C07234=1040.428,9.851,-82.657,169.408,37.411,157.036
C07235=1040.433,10.101,-82.672,169.410,37.411,157.036
C07236=1040.440,10.351,-82.687,169.412,37.412,157.036
C07237=1040.446,10.600,-82.703,169.414,37.412,157.036
C07238=1040.453,10.849,-82.718,169.416,37.413,157.036
C07239=1040.460,11.098,-82.734,169.417,37.414,157.036
C07240=1040.466,11.348,-82.749,169.419,37.414,157.037
C07241=1040.472,11.598,-82.764,169.421,37.415,157.037
C07242=1040.479,11.847,-82.779,169.423,37.415,157.037
C07243=1040.485,12.097,-82.795,169.426,37.416,157.037
C07244=1040.492,12.382,-82.812,169.429,37.416,157.037
C07245=1040.500,12.667,-82.830,169.431,37.418,157.037
C07246=1040.507,12.952,-82.848,169.433,37.418,157.037
C07247=1040.514,13.238,-82.865,169.435,37.419,157.038
C07248=1040.521,13.487,-82.880,169.437,37.419,157.038
C07249=1040.528,13.737,-82.895,169.439,37.420,157.038
C07250=1040.534,13.986,-82.911,169.441,37.421,157.038
C07251=1040.540,14.236,-82.927,169.443,37.421,157.038
C07252=1040.547,14.485,-82.942,169.446,37.422,157.038
C07253=1040.553,14.735,-82.957,169.448,37.423,157.039
C07254=1040.559,14.984,-82.973,169.450,37.424,157.039
C07255=1040.566,15.233,-82.989,169.452,37.424,157.039
C07256=1040.574,15.563,-83.009,169.454,37.425,157.039
C07257=1040.582,15.892,-83.031,169.457,37.426,157.039
C07258=1040.590,16.223,-83.051,169.459,37.427,157.039
C07259=1040.599,16.552,-83.071,169.463,37.428,157.040
C07260=1040.605,16.802,-83.087,169.465,37.429,157.040
C07261=1040.611,17.051,-83.103,169.467,37.430,157.040
C07262=1040.618,17.301,-83.118,169.468,37.430,157.040
C07263=1040.624,17.550,-83.134,169.470,37.431,157.040
C07264=1040.630,17.799,-83.150,169.472,37.432,157.040
C07265=1040.637,18.049,-83.165,169.474,37.433,157.041
C07266=1040.643,18.298,-83.181,169.476,37.433,157.041
C07267=1040.649,18.547,-83.197,169.478,37.434,157.041
C07268=1040.656,18.797,-83.212,169.480,37.434,157.041
C07269=1040.662,19.047,-83.228,169.483,37.435,157.041
C07270=1040.669,19.296,-83.244,169.485,37.436,157.041
C07271=1040.675,19.546,-83.260,169.487,37.437,157.041
C07272=1040.681,19.795,-83.275,169.489,37.437,157.042
C07273=1040.688,20.044,-83.291,169.490,37.438,157.042
C07274=1040.694,20.293,-83.307,169.492,37.439,157.042
C07275=1040.700,20.543,-83.323,169.494,37.440,157.042
C07276=1040.706,20.792,-83.338,169.496,37.440,157.042
C07277=1040.712,21.041,-83.355,169.498,37.441,157.042
C07278=1040.720,21.291,-83.371,169.501,37.442,157.042
C07279=1040.725,21.541,-83.386,169.503,37.443,157.043
C07280=1040.732,21.790,-83.402,169.505,37.443,157.043
C07281=1040.738,22.040,-83.418,169.506,37.444,157.043
C07282=1040.745,22.289,-83.434,169.508,37.445,157.043
C07283=1040.750,22.538,-83.450,169.510,37.446,157.043
C07284=1040.757,22.787,-83.466,169.512,37.447,157.043
C07285=1040.763,23.037,-83.481,169.514,37.447,157.044
C07286=1040.770,23.287,-83.497,169.517,37.448,157.044
C07287=1040.776,23.536,-83.514,169.519,37.449,157.044
C07288=1040.782,23.785,-83.530,169.521,37.450,157.044
C07289=1040.789,24.034,-83.545,169.523,37.450,157.044
C07290=1040.795,24.284,-83.562,169.524,37.451,157.044
C07291=1040.801,24.533,-83.577,169.526,37.452,157.045
C07292=1040.808,24.783,-83.593,169.528,37.453,157.045
C07293=1040.814,25.032,-83.609,169.530,37.453,157.045
C07294=1040.820,25.282,-83.625,169.532,37.454,157.045
C07295=1040.827,25.531,-83.641,169.535,37.455,157.045
C07296=1040.833,25.780,-83.657,169.537,37.456,157.045
C07297=1040.839,26.030,-83.674,169.539,37.456,157.046
C07298=1040.846,26.279,-83.689,169.540,37.457,157.046
C07299=1040.852,26.529,-83.706,169.542,37.458,157.046
C07300=1040.859,26.778,-83.721,169.544,37.459,157.046
C07301=1040.865,27.027,-83.738,169.546,37.459,157.046
C07302=1040.871,27.277,-83.754,169.548,37.460,157.046
C07303=1040.878,27.526,-83.770,169.551,37.461,157.047
C07304=1040.883,27.754,-83.785,169.552,37.462,157.047
C07305=1040.889,27.982,-83.799,169.554,37.462,157.047
C07306=1040.895,28.210,-83.814,169.556,37.463,157.047
C07307=1040.901,28.438,-83.829,169.558,37.463,157.047
C07308=1040.906,28.666,-83.843,169.559,37.464,157.047
C07309=1040.912,28.893,-83.858,169.561,37.465,157.047
C07310=1040.918,29.122,-83.873,169.563,37.466,157.048
C07311=1040.924,29.350,-83.888,169.564,37.466,157.048
C07312=1040.930,29.599,-83.905,169.566,37.467,157.048
C07313=1040.936,29.848,-83.921,169.569,37.468,157.048
C07314=1040.942,30.097,-83.937,169.571,37.469,157.048
C07315=1040.949,30.347,-83.953,169.573,37.469,157.048
C07316=1040.955,30.597,-83.969,169.575,37.471,157.049
C07317=1040.961,30.846,-83.986,169.576,37.471,157.049
C07318=1040.967,31.095,-84.002,169.578,37.472,157.049
C07319=1040.974,31.345,-84.019,169.580,37.473,157.049
C07320=1040.980,31.594,-84.034,169.583,37.474,157.049
C07321=1040.987,31.843,-84.051,169.585,37.474,157.049
C07322=1040.993,32.092,-84.068,169.587,37.475,157.050
C07323=1040.999,32.342,-84.084,169.588,37.476,157.050
C07324=1041.006,32.592,-84.100,169.590,37.477,157.050
C07325=1041.012,32.841,-84.116,169.592,37.478,157.050
C07326=1041.018,33.091,-84.133,169.594,37.478,157.050
C07327=1041.025,33.340,-84.150,169.596,37.479,157.050
C07328=1041.031,33.589,-84.166,169.599,37.480,157.051
C07329=1041.037,33.838,-84.182,169.600,37.481,157.051
C07330=1041.044,34.088,-84.198,169.602,37.481,157.051
C07331=1041.050,34.337,-84.214,169.604,37.483,157.051
C07332=1041.056,34.586,-84.231,169.606,37.483,157.051
C07333=1041.063,34.836,-84.248,169.608,37.484,157.051
C07334=1041.069,35.086,-84.264,169.610,37.485,157.052
C07335=1041.075,35.335,-84.280,169.612,37.486,157.052
C07336=1041.082,35.584,-84.297,169.613,37.486,157.052
C07337=1041.088,35.833,-84.314,169.616,37.487,157.052
C07338=1041.094,36.083,-84.330,169.618,37.488,157.052
C07339=1041.101,36.333,-84.346,169.620,37.489,157.052
C07340=1041.107,36.582,-84.363,169.622,37.489,157.053
C07341=1041.114,36.831,-84.379,169.624,37.490,157.053
C07342=1041.120,37.081,-84.396,169.625,37.491,157.053
C07343=1041.126,37.330,-84.412,169.627,37.492,157.053
C07344=1041.133,37.579,-84.429,169.630,37.493,157.053
C07345=1041.139,37.829,-84.446,169.632,37.493,157.053
C07346=1041.145,38.077,-84.463,169.634,37.494,157.054
C07347=1041.152,38.328,-84.479,169.635,37.495,157.054
C07348=1041.158,38.577,-84.495,169.637,37.496,157.054
C07349=1041.164,38.826,-84.512,169.639,37.497,157.054
C07350=1041.170,39.076,-84.529,169.641,37.498,157.054
C07351=1041.176,39.325,-84.545,169.643,37.499,157.055
C07352=1041.183,39.574,-84.562,169.645,37.499,157.055
C07353=1041.189,39.824,-84.579,169.647,37.500,157.055
C07354=1041.195,40.072,-84.596,169.649,37.501,157.055
C07355=1041.202,40.323,-84.612,169.651,37.502,157.055
C07356=1041.208,40.571,-84.629,169.653,37.503,157.056
C07357=1041.214,40.821,-84.646,169.655,37.504,157.056
C07358=1041.220,41.071,-84.663,169.656,37.504,157.056
C07359=1041.226,41.320,-84.680,169.658,37.506,157.056
C07360=1041.233,41.570,-84.696,169.661,37.506,157.056
C07361=1041.239,41.818,-84.713,169.663,37.507,157.056
C07362=1041.245,42.068,-84.730,169.665,37.508,157.057
C07363=1041.252,42.317,-84.747,169.666,37.509,157.057
C07364=1041.258,42.567,-84.763,169.668,37.510,157.057
C07365=1041.265,42.816,-84.781,169.670,37.510,157.057
C07366=1041.271,43.065,-84.797,169.672,37.512,157.057
C07367=1041.277,43.314,-84.814,169.675,37.512,157.057
C07368=1041.284,43.564,-84.831,169.676,37.513,157.058
C07369=1041.289,43.813,-84.848,169.678,37.514,157.058
C07370=1041.296,44.063,-84.865,169.680,37.515,157.058
C07371=1041.302,44.312,-84.882,169.682,37.516,157.058
C07372=1041.309,44.598,-84.902,169.684,37.517,157.058
C07373=1041.316,44.885,-84.921,169.686,37.518,157.059
C07374=1041.323,45.172,-84.940,169.689,37.519,157.059
C07375=1041.330,45.458,-84.961,169.691,37.520,157.059
C07376=1041.336,45.708,-84.977,169.693,37.521,157.059
C07377=1041.342,45.956,-84.994,169.694,37.522,157.059
C07378=1041.349,46.206,-85.012,169.696,37.523,157.060
C07379=1041.355,46.456,-85.028,169.698,37.524,157.060
C07380=1041.361,46.705,-85.046,169.700,37.525,157.060
C07381=1041.367,46.954,-85.063,169.703,37.525,157.060
C07382=1041.373,47.204,-85.080,169.704,37.527,157.060
C07383=1041.380,47.453,-85.097,169.706,37.527,157.061
C07384=1041.386,47.703,-85.115,169.708,37.528,157.061
C07385=1041.392,47.951,-85.132,169.710,37.529,157.061
C07386=1041.399,48.201,-85.148,169.711,37.530,157.061
C07387=1041.404,48.450,-85.166,169.713,37.531,157.061
C07388=1041.410,48.699,-85.183,169.716,37.532,157.062
C07389=1041.417,48.949,-85.199,169.718,37.533,157.062
C07390=1041.422,49.198,-85.217,169.719,37.534,157.062
C07391=1041.429,49.448,-85.234,169.721,37.535,157.062
C07392=1041.436,49.696,-85.251,169.723,37.536,157.062
C07393=1041.441,49.947,-85.268,169.725,37.536,157.063
C07394=1041.448,50.195,-85.285,169.727,37.538,157.063
C07395=1041.455,50.445,-85.303,169.729,37.538,157.063
C07396=1041.460,50.694,-85.320,169.731,37.539,157.063
C07397=1041.467,50.943,-85.338,169.733,37.540,157.063
C07398=1041.473,51.193,-85.354,169.735,37.541,157.064
C07399=1041.479,51.442,-85.372,169.736,37.542,157.064
C07400=1041.486,51.692,-85.389,169.738,37.543,157.064
C07401=1041.492,51.941,-85.406,169.740,37.544,157.064
C07402=1041.498,52.190,-85.424,169.743,37.545,157.064
C07403=1041.504,52.439,-85.441,169.745,37.545,157.064
C07404=1041.510,52.689,-85.458,169.746,37.547,157.065
C07405=1041.517,52.938,-85.475,169.748,37.547,157.065
C07406=1041.523,53.188,-85.493,169.750,37.548,157.065
C07407=1041.529,53.437,-85.510,169.752,37.549,157.065
C07408=1041.536,53.686,-85.528,169.753,37.550,157.065
C07409=1041.543,53.935,-85.545,169.756,37.551,157.066
C07410=1041.548,54.185,-85.562,169.758,37.551,157.066
C07411=1041.555,54.434,-85.580,169.760,37.553,157.066
C07412=1041.561,54.683,-85.597,169.762,37.553,157.066
C07413=1041.567,54.933,-85.614,169.763,37.554,157.066
C07414=1041.574,55.182,-85.631,169.765,37.555,157.066
C07415=1041.579,55.432,-85.649,169.767,37.556,157.067
C07416=1041.586,55.681,-85.666,169.769,37.557,157.067
C07417=1041.593,55.930,-85.683,169.771,37.558,157.067
C07418=1041.599,56.179,-85.701,169.773,37.559,157.067
C07419=1041.606,56.429,-85.718,169.775,37.559,157.067
C07420=1041.612,56.678,-85.735,169.777,37.560,157.068
C07421=1041.618,56.927,-85.753,169.779,37.561,157.068
C07422=1041.625,57.177,-85.771,169.780,37.562,157.068
C07423=1041.630,57.426,-85.788,169.782,37.563,157.068
C07424=1041.637,57.675,-85.806,169.785,37.564,157.068
C07425=1041.643,57.924,-85.823,169.787,37.565,157.069
C07426=1041.650,58.174,-85.840,169.789,37.566,157.069
C07427=1041.656,58.423,-85.858,169.790,37.566,157.069
C07428=1041.662,58.672,-85.875,169.792,37.567,157.069
C07429=1041.669,58.922,-85.893,169.794,37.568,157.069
C07430=1041.676,59.171,-85.910,169.796,37.569,157.069
C07431=1041.682,59.421,-85.928,169.798,37.570,157.070
C07432=1041.688,59.669,-85.945,169.800,37.571,157.070
C07433=1041.694,59.919,-85.963,169.802,37.571,157.070
C07434=1041.701,60.169,-85.980,169.804,37.572,157.070
C07435=1041.707,60.417,-85.997,169.806,37.573,157.070
C07436=1041.715,60.704,-86.018,169.808,37.574,157.071
C07437=1041.722,60.990,-86.037,169.810,37.575,157.071
C07438=1041.730,61.276,-86.059,169.813,37.576,157.071
C07439=1041.737,61.562,-86.078,169.815,37.577,157.071
C07440=1041.743,61.812,-86.096,169.817,37.578,157.071
C07441=1041.750,62.061,-86.114,169.818,37.579,157.072
C07442=1041.756,62.311,-86.131,169.820,37.580,157.072
C07443=1041.762,62.560,-86.149,169.822,37.580,157.072
C07444=1041.769,62.809,-86.166,169.824,37.581,157.072
C07445=1041.775,63.059,-86.184,169.827,37.582,157.072
C07446=1041.782,63.308,-86.202,169.828,37.583,157.073
C07447=1041.788,63.556,-86.219,169.830,37.584,157.073
C07448=1041.794,63.806,-86.237,169.832,37.584,157.073
C07449=1041.801,64.056,-86.255,169.834,37.586,157.073
C07450=1041.807,64.305,-86.272,169.835,37.587,157.073
C07451=1041.813,64.554,-86.290,169.837,37.587,157.073
C07452=1041.819,64.803,-86.308,169.840,37.589,157.074
C07453=1041.826,65.053,-86.326,169.842,37.589,157.074
C07454=1041.832,65.303,-86.344,169.843,37.590,157.074
C07455=1041.838,65.551,-86.362,169.845,37.591,157.074
C07456=1041.845,65.800,-86.379,169.847,37.592,157.074
C07457=1041.851,66.050,-86.397,169.849,37.593,157.075
C07458=1041.858,66.299,-86.416,169.850,37.594,157.075
C07459=1041.864,66.548,-86.433,169.853,37.595,157.075
C07460=1041.870,66.798,-86.451,169.855,37.596,157.075
C07461=1041.876,67.047,-86.469,169.857,37.596,157.075
C07462=1041.883,67.297,-86.487,169.859,37.598,157.076
C07463=1041.889,67.545,-86.504,169.860,37.599,157.076
C07464=1041.895,67.794,-86.523,169.862,37.599,157.076
C07465=1041.901,68.044,-86.541,169.864,37.601,157.076
C07466=1041.907,68.294,-86.559,169.867,37.601,157.076
C07467=1041.914,68.542,-86.576,169.868,37.602,157.077
C07468=1041.920,68.792,-86.594,169.870,37.603,157.077
C07469=1041.926,69.041,-86.612,169.872,37.604,157.077
C07470=1041.933,69.291,-86.631,169.874,37.605,157.077
C07471=1041.940,69.540,-86.648,169.875,37.606,157.077
C07472=1041.945,69.788,-86.667,169.878,37.607,157.078
C07473=1041.951,70.038,-86.685,169.880,37.608,157.078
C07474=1041.958,70.287,-86.703,169.882,37.609,157.078
C07475=1041.964,70.537,-86.721,169.883,37.610,157.078
C07476=1041.970,70.787,-86.739,169.885,37.611,157.078
C07477=1041.976,71.035,-86.757,169.887,37.612,157.079
C07478=1041.983,71.285,-86.775,169.889,37.613,157.079
C07479=1041.989,71.534,-86.793,169.891,37.614,157.079
C07480=1041.995,71.784,-86.811,169.893,37.614,157.079
C07481=1042.002,72.033,-86.830,169.895,37.616,157.079
C07482=1042.007,72.282,-86.847,169.897,37.617,157.080
C07483=1042.014,72.531,-86.866,169.898,37.617,157.080
C07484=1042.020,72.780,-86.885,169.900,37.619,157.080
C07485=1042.026,73.030,-86.903,169.902,37.619,157.080
C07486=1042.033,73.279,-86.921,169.905,37.620,157.080
C07487=1042.038,73.528,-86.939,169.906,37.622,157.081
C07488=1042.045,73.777,-86.958,169.908,37.622,157.081
C07489=1042.052,74.026,-86.975,169.910,37.623,157.081
C07490=1042.058,74.275,-86.994,169.911,37.624,157.081
C07491=1042.064,74.525,-87.012,169.913,37.625,157.081
C07492=1042.070,74.774,-87.030,169.916,37.626,157.082
C07493=1042.077,75.023,-87.049,169.918,37.627,157.082
C07494=1042.082,75.273,-87.066,169.920,37.628,157.082
C07495=1042.089,75.522,-87.085,169.921,37.629,157.082
C07496=1042.095,75.771,-87.104,169.923,37.630,157.083
C07497=1042.101,76.020,-87.122,169.925,37.631,157.083
C07498=1042.108,76.270,-87.140,169.928,37.632,157.083
C07499=1042.114,76.519,-87.158,169.929,37.633,157.083
C07500=1042.122,76.805,-87.179,169.931,37.634,157.083
C07501=1042.128,77.091,-87.200,169.933,37.635,157.084
C07502=1042.136,77.377,-87.222,169.935,37.636,157.084
C07503=1042.143,77.663,-87.243,169.937,37.637,157.084
C07504=1042.149,77.912,-87.261,169.939,37.638,157.084
C07505=1042.155,78.162,-87.279,169.942,37.639,157.084
C07506=1042.162,78.411,-87.298,169.944,37.640,157.085
C07507=1042.168,78.660,-87.316,169.945,37.641,157.085
C07508=1042.174,78.909,-87.335,169.947,37.642,157.085
C07509=1042.180,79.159,-87.354,169.949,37.643,157.085
C07510=1042.186,79.408,-87.372,169.950,37.644,157.085
C07511=1042.193,79.657,-87.391,169.953,37.645,157.086
C07512=1042.199,79.907,-87.409,169.955,37.646,157.086
C07513=1042.205,80.155,-87.427,169.957,37.647,157.086
C07514=1042.210,80.405,-87.447,169.958,37.648,157.086
C07515=1042.217,80.654,-87.465,169.960,37.649,157.087
C07516=1042.223,80.903,-87.484,169.963,37.650,157.087
C07517=1042.229,81.153,-87.502,169.965,37.651,157.087
C07518=1042.236,81.402,-87.520,169.966,37.652,157.087
C07519=1042.242,81.651,-87.540,169.968,37.653,157.088
C07520=1042.248,81.900,-87.558,169.970,37.654,157.088
C07521=1042.254,82.150,-87.577,169.972,37.655,157.088
C07522=1042.261,82.399,-87.596,169.973,37.656,157.088
C07523=1042.267,82.648,-87.614,169.976,37.657,157.088
C07524=1042.273,82.897,-87.634,169.978,37.658,157.089
C07525=1042.279,83.147,-87.651,169.980,37.659,157.089
C07526=1042.285,83.396,-87.670,169.981,37.660,157.089
C07527=1042.291,83.644,-87.688,169.983,37.661,157.089
C07528=1042.298,83.894,-87.707,169.985,37.662,157.089
C07529=1042.303,84.143,-87.726,169.988,37.663,157.090
C07530=1042.310,84.392,-87.745,169.989,37.664,157.090
C07531=1042.316,84.641,-87.764,169.991,37.665,157.090
C07532=1042.323,84.890,-87.782,169.993,37.666,157.090
C07533=1042.329,85.140,-87.801,169.995,37.667,157.091
C07534=1042.335,85.389,-87.820,169.996,37.668,157.091
C07535=1042.341,85.638,-87.839,169.999,37.669,157.091
C07536=1042.348,85.887,-87.857,170.001,37.670,157.091
C07537=1042.354,86.136,-87.876,170.003,37.671,157.091
C07538=1042.360,86.386,-87.895,170.004,37.672,157.092
C07539=1042.366,86.635,-87.914,170.006,37.673,157.092
C07540=1042.373,86.884,-87.933,170.008,37.674,157.092
C07541=1042.380,87.134,-87.952,170.011,37.675,157.092
C07542=1042.386,87.383,-87.970,170.012,37.676,157.092
C07543=1042.392,87.632,-87.990,170.014,37.677,157.093
C07544=1042.398,87.882,-88.008,170.016,37.678,157.093
C07545=1042.405,88.131,-88.027,170.018,37.679,157.093
C07546=1042.411,88.380,-88.045,170.019,37.680,157.093
C07547=1042.417,88.629,-88.065,170.021,37.681,157.093
C07548=1042.423,88.878,-88.083,170.024,37.681,157.094
C07549=1042.430,89.127,-88.102,170.026,37.683,157.094
C07550=1042.436,89.377,-88.121,170.027,37.684,157.094
C07551=1042.442,89.626,-88.140,170.029,37.684,157.094
C07552=1042.448,89.875,-88.159,170.031,37.686,157.095
C07553=1042.455,90.124,-88.177,170.033,37.687,157.095
C07554=1042.460,90.374,-88.196,170.035,37.687,157.095
C07555=1042.467,90.622,-88.216,170.037,37.689,157.095
C07556=1042.473,90.872,-88.235,170.039,37.690,157.095
C07557=1042.480,91.121,-88.254,170.041,37.691,157.096
C07558=1042.485,91.371,-88.273,170.042,37.692,157.096
C07559=1042.492,91.620,-88.292,170.044,37.693,157.096
C07560=1042.498,91.869,-88.312,170.047,37.694,157.096
C07561=1042.504,92.118,-88.331,170.049,37.695,157.097
C07562=1042.510,92.367,-88.350,170.050,37.696,157.097
C07563=1042.516,92.616,-88.368,170.052,37.697,157.097
C07564=1042.524,92.902,-88.391,170.054,37.698,157.097
C07565=1042.531,93.189,-88.412,170.057,37.699,157.097
C07566=1042.537,93.474,-88.435,170.059,37.701,157.098
C07567=1042.544,93.760,-88.457,170.061,37.702,157.098
C07568=1042.551,94.009,-88.475,170.063,37.703,157.098
C07569=1042.557,94.259,-88.496,170.065,37.704,157.099
C07570=1042.564,94.508,-88.514,170.066,37.705,157.099
C07571=1042.569,94.757,-88.534,170.069,37.706,157.099
C07572=1042.576,95.006,-88.552,170.071,37.707,157.099
C07573=1042.582,95.255,-88.572,170.073,37.708,157.099
C07574=1042.588,95.504,-88.591,170.074,37.709,157.100
C07575=1042.594,95.754,-88.610,170.076,37.710,157.100
C07576=1042.600,96.003,-88.630,170.078,37.711,157.100
C07577=1042.607,96.252,-88.649,170.081,37.712,157.100
C07578=1042.613,96.502,-88.668,170.082,37.713,157.100
C07579=1042.619,96.750,-88.688,170.084,37.714,157.101
C07580=1042.625,97.000,-88.707,170.086,37.716,157.101
C07581=1042.631,97.249,-88.725,170.088,37.716,157.101
C07582=1042.637,97.498,-88.745,170.089,37.717,157.101
C07583=1042.644,97.748,-88.764,170.092,37.719,157.102
C07584=1042.650,97.996,-88.784,170.094,37.719,157.102
C07585=1042.657,98.246,-88.803,170.096,37.720,157.102
C07586=1042.662,98.495,-88.822,170.098,37.722,157.102
C07587=1042.668,98.744,-88.842,170.099,37.723,157.103
C07588=1042.675,98.993,-88.861,170.101,37.723,157.103
C07589=1042.682,99.242,-88.881,170.104,37.725,157.103
C07590=1042.688,99.492,-88.900,170.106,37.726,157.103
C07591=1042.694,99.740,-88.920,170.107,37.726,157.103
C07592=1042.700,99.989,-88.938,170.109,37.728,157.104
C07593=1042.706,100.239,-88.958,170.111,37.729,157.104
C07594=1042.713,100.488,-88.978,170.113,37.729,157.104
C07595=1042.719,100.738,-88.997,170.116,37.730,157.104
C07596=1042.725,100.986,-89.017,170.117,37.732,157.104
C07597=1042.731,101.235,-89.037,170.119,37.733,157.105
C07598=1042.737,101.485,-89.056,170.121,37.734,157.105
C07599=1042.743,101.734,-89.076,170.123,37.735,157.105
C07600=1042.750,101.983,-89.095,170.125,37.736,157.105
C07601=1042.756,102.232,-89.115,170.127,37.737,157.106
C07602=1042.761,102.481,-89.134,170.129,37.738,157.106
C07603=1042.767,102.730,-89.154,170.131,37.739,157.106
C07604=1042.774,102.980,-89.174,170.132,37.741,157.106
C07605=1042.780,103.229,-89.193,170.135,37.742,157.107
C07606=1042.786,103.478,-89.213,170.137,37.742,157.107
C07607=1042.792,103.727,-89.232,170.139,37.744,157.107
C07608=1042.798,103.976,-89.252,170.140,37.745,157.107
C07609=1042.805,104.225,-89.272,170.142,37.746,157.108
C07610=1042.811,104.475,-89.291,170.144,37.747,157.108
C07611=1042.817,104.723,-89.311,170.147,37.748,157.108
C07612=1042.823,104.972,-89.331,170.148,37.749,157.108
C07613=1042.829,105.222,-89.351,170.150,37.750,157.108
C07614=1042.835,105.471,-89.371,170.152,37.751,157.109
C07615=1042.841,105.720,-89.391,170.154,37.753,157.109
C07616=1042.848,105.969,-89.409,170.155,37.753,157.109
C07617=1042.854,106.219,-89.430,170.158,37.754,157.109
C07618=1042.860,106.467,-89.449,170.160,37.756,157.110
C07619=1042.866,106.717,-89.469,170.162,37.757,157.110
C07620=1042.873,106.966,-89.489,170.164,37.758,157.110
C07621=1042.879,107.215,-89.509,170.165,37.759,157.110
C07622=1042.885,107.464,-89.528,170.168,37.760,157.111
C07623=1042.891,107.713,-89.548,170.170,37.761,157.111
C07624=1042.898,107.963,-89.568,170.172,37.762,157.111
C07625=1042.904,108.211,-89.588,170.174,37.763,157.111
C07626=1042.909,108.461,-89.607,170.175,37.764,157.111
C07627=1042.916,108.710,-89.627,170.177,37.765,157.112
C07628=1042.923,108.996,-89.650,170.180,37.766,157.112
C07629=1042.930,109.282,-89.673,170.182,37.767,157.112
C07630=1042.938,109.568,-89.695,170.184,37.769,157.113
C07631=1042.944,109.854,-89.718,170.186,37.770,157.113
C07632=1042.951,110.103,-89.738,170.188,37.771,157.113
C07633=1042.957,110.352,-89.758,170.191,37.772,157.113
C07634=1042.963,110.602,-89.779,170.193,37.773,157.114
C07635=1042.970,110.850,-89.798,170.195,37.774,157.114
C07636=1042.975,111.099,-89.819,170.196,37.775,157.114
C07637=1042.982,111.349,-89.838,170.198,37.776,157.114
C07638=1042.988,111.598,-89.858,170.201,37.778,157.114
C07639=1042.994,111.847,-89.878,170.203,37.779,157.115
C07640=1043.000,112.097,-89.898,170.204,37.780,157.115
C07641=1043.006,112.345,-89.918,170.206,37.781,157.115
C07642=1043.012,112.594,-89.938,170.208,37.782,157.115
C07643=1043.019,112.844,-89.959,170.210,37.783,157.116
C07644=1043.025,113.093,-89.979,170.213,37.784,157.116
C07645=1043.031,113.341,-89.999,170.214,37.785,157.116
C07646=1043.037,113.591,-90.019,170.216,37.786,157.116
C07647=1043.043,113.840,-90.039,170.218,37.788,157.117
C07648=1043.049,114.089,-90.059,170.220,37.789,157.117
C07649=1043.056,114.338,-90.079,170.223,37.790,157.117
C07650=1043.061,114.587,-90.100,170.224,37.791,157.117
C07651=1043.067,114.836,-90.120,170.226,37.792,157.118
C07652=1043.074,115.085,-90.140,170.228,37.793,157.118
C07653=1043.079,115.335,-90.161,170.230,37.794,157.118
C07654=1043.085,115.583,-90.181,170.232,37.795,157.118
C07655=1043.092,115.833,-90.201,170.234,37.797,157.119
C07656=1043.098,116.082,-90.221,170.236,37.798,157.119
C07657=1043.104,116.332,-90.242,170.238,37.799,157.119
C07658=1043.110,116.580,-90.262,170.240,37.800,157.119
C07659=1043.116,116.829,-90.282,170.242,37.801,157.120
C07660=1043.122,117.078,-90.303,170.244,37.803,157.120
C07661=1043.128,117.327,-90.323,170.246,37.804,157.120
C07662=1043.134,117.576,-90.343,170.248,37.805,157.120
C07663=1043.140,117.826,-90.364,170.249,37.806,157.121
C07664=1043.146,118.075,-90.384,170.252,37.807,157.121
C07665=1043.152,118.324,-90.404,170.254,37.809,157.121
C07666=1043.158,118.573,-90.424,170.256,37.810,157.121
C07667=1043.164,118.821,-90.445,170.258,37.811,157.122
C07668=1043.170,119.071,-90.466,170.259,37.812,157.122
C07669=1043.176,119.320,-90.486,170.262,37.813,157.122
C07670=1043.183,119.569,-90.506,170.264,37.814,157.123
C07671=1043.188,119.818,-90.527,170.266,37.816,157.123
C07672=1043.195,120.067,-90.548,170.268,37.817,157.123
C07673=1043.201,120.316,-90.568,170.269,37.818,157.123
C07674=1043.206,120.565,-90.588,170.271,37.819,157.123
C07675=1043.213,120.815,-90.609,170.274,37.820,157.124
C07676=1043.219,121.063,-90.629,170.276,37.821,157.124
C07677=1043.225,121.313,-90.650,170.278,37.822,157.124
C07678=1043.231,121.562,-90.670,170.280,37.823,157.124
C07679=1043.238,121.811,-90.691,170.282,37.825,157.125
C07680=1043.244,122.059,-90.711,170.284,37.826,157.125
C07681=1043.250,122.309,-90.732,170.286,37.827,157.125
C07682=1043.256,122.558,-90.752,170.288,37.828,157.126
C07683=1043.262,122.808,-90.772,170.290,37.829,157.126
C07684=1043.268,123.056,-90.794,170.292,37.831,157.126
C07685=1043.275,123.306,-90.814,170.294,37.832,157.126
C07686=1043.281,123.554,-90.834,170.296,37.833,157.127
C07687=1043.287,123.804,-90.856,170.298,37.834,157.127
C07688=1043.293,124.052,-90.876,170.300,37.835,157.127
C07689=1043.299,124.302,-90.896,170.302,37.836,157.127
C07690=1043.305,124.550,-90.917,170.304,37.837,157.127
C07691=1043.311,124.800,-90.937,170.306,37.838,157.128
C07692=1043.318,125.085,-90.961,170.308,37.839,157.128
C07693=1043.326,125.371,-90.985,170.311,37.841,157.128
C07694=1043.333,125.657,-91.008,170.314,37.842,157.129
C07695=1043.340,125.944,-91.032,170.316,37.844,157.129
C07696=1043.346,126.192,-91.053,170.318,37.845,157.129
C07697=1043.353,126.442,-91.074,170.319,37.846,157.129
C07698=1043.359,126.690,-91.094,170.321,37.847,157.130
C07699=1043.365,126.940,-91.115,170.324,37.848,157.130
C07700=1043.371,127.188,-91.135,170.326,37.849,157.130
C07701=1043.378,127.437,-91.156,170.328,37.850,157.130
C07702=1043.383,127.687,-91.177,170.330,37.851,157.131
C07703=1043.390,127.935,-91.198,170.332,37.852,157.131
C07704=1043.396,128.185,-91.219,170.334,37.854,157.131
C07705=1043.402,128.434,-91.239,170.336,37.855,157.131
C07706=1043.409,128.683,-91.260,170.338,37.856,157.132
C07707=1043.414,128.933,-91.281,170.340,37.857,157.132
C07708=1043.421,129.181,-91.301,170.342,37.858,157.132
C07709=1043.427,129.430,-91.322,170.345,37.859,157.132
C07710=1043.433,129.680,-91.343,170.347,37.861,157.133
C07711=1043.439,129.928,-91.363,170.349,37.862,157.133
C07712=1043.446,130.177,-91.384,170.350,37.862,157.133
C07713=1043.452,130.426,-91.406,170.352,37.864,157.133
C07714=1043.458,130.675,-91.426,170.354,37.865,157.134
C07715=1043.465,130.924,-91.448,170.357,37.866,157.134
C07716=1043.471,131.173,-91.468,170.359,37.867,157.134
C07717=1043.477,131.422,-91.489,170.361,37.868,157.134
C07718=1043.483,131.672,-91.510,170.363,37.869,157.135
C07719=1043.489,131.921,-91.531,170.365,37.871,157.135
C07720=1043.495,132.170,-91.552,170.367,37.872,157.135
C07721=1043.502,132.419,-91.573,170.369,37.873,157.135
C07722=1043.507,132.668,-91.594,170.371,37.874,157.136
C07723=1043.513,132.917,-91.616,170.373,37.875,157.136
C07724=1043.519,133.166,-91.636,170.376,37.877,157.136
C07725=1043.526,133.415,-91.657,170.378,37.878,157.137
C07726=1043.532,133.664,-91.679,170.380,37.879,157.137
C07727=1043.538,133.912,-91.700,170.381,37.881,157.137
C07728=1043.544,134.162,-91.720,170.383,37.882,157.137
C07729=1043.550,134.411,-91.742,170.386,37.883,157.138
C07730=1043.556,134.660,-91.763,170.388,37.884,157.138
C07731=1043.563,134.909,-91.784,170.390,37.885,157.138
C07732=1043.568,135.159,-91.805,170.392,37.887,157.138
C07733=1043.575,135.407,-91.826,170.394,37.888,157.139
C07734=1043.581,135.656,-91.848,170.397,37.889,157.139
C07735=1043.587,135.905,-91.869,170.398,37.890,157.139
C07736=1043.593,136.154,-91.889,170.400,37.891,157.140
C07737=1043.599,136.403,-91.911,170.402,37.893,157.140
C07738=1043.605,136.652,-91.933,170.404,37.894,157.140
C07739=1043.612,136.901,-91.954,170.407,37.895,157.140
C07740=1043.618,137.150,-91.975,170.409,37.896,157.141
C07741=1043.624,137.400,-91.996,170.411,37.897,157.141
C07742=1043.630,137.649,-92.017,170.413,37.898,157.141
C07743=1043.636,137.897,-92.038,170.416,37.900,157.141
C07744=1043.642,138.146,-92.060,170.417,37.901,157.142
C07745=1043.648,138.395,-92.081,170.419,37.902,157.142
C07746=1043.655,138.645,-92.103,170.421,37.904,157.142
C07747=1043.660,138.893,-92.124,170.423,37.905,157.143
C07748=1043.667,139.142,-92.145,170.426,37.906,157.143
C07749=1043.673,139.391,-92.167,170.428,37.907,157.143
C07750=1043.679,139.641,-92.188,170.430,37.908,157.143
C07751=1043.685,139.890,-92.209,170.432,37.910,157.144
C07752=1043.691,140.139,-92.231,170.434,37.911,157.144
C07753=1043.697,140.388,-92.252,170.436,37.912,157.144
C07754=1043.703,140.637,-92.274,170.438,37.913,157.144
C07755=1043.709,140.886,-92.295,170.440,37.915,157.145
C07756=1043.717,141.171,-92.320,170.442,37.916,157.145
C07757=1043.723,141.457,-92.344,170.446,37.917,157.145
C07758=1043.730,141.743,-92.370,170.448,37.919,157.146
C07759=1043.737,142.027,-92.394,170.450,37.920,157.146
C07760=1043.744,142.277,-92.416,170.452,37.922,157.146
C07761=1043.750,142.526,-92.437,170.455,37.923,157.147
C07762=1043.756,142.775,-92.459,170.457,37.924,157.147
C07763=1043.761,143.024,-92.480,170.459,37.926,157.147
C07764=1043.768,143.273,-92.502,170.461,37.927,157.147
C07765=1043.774,143.522,-92.523,170.464,37.928,157.148
C07766=1043.780,143.771,-92.545,170.465,37.929,157.148
C07767=1043.786,144.020,-92.567,170.467,37.931,157.148
C07768=1043.792,144.269,-92.588,170.469,37.932,157.149
C07769=1043.798,144.518,-92.610,170.471,37.933,157.149
C07770=1043.804,144.767,-92.632,170.474,37.934,157.149
C07771=1043.810,145.016,-92.654,170.476,37.936,157.149
C07772=1043.817,145.265,-92.675,170.478,37.937,157.150
C07773=1043.823,145.514,-92.697,170.480,37.938,157.150
C07774=1043.828,145.763,-92.718,170.482,37.939,157.150
C07775=1043.835,146.012,-92.740,170.485,37.941,157.151
C07776=1043.841,146.261,-92.761,170.487,37.942,157.151
C07777=1043.847,146.510,-92.784,170.489,37.943,157.151
C07778=1043.854,146.759,-92.805,170.491,37.944,157.151
C07779=1043.860,147.008,-92.826,170.494,37.946,157.152
C07780=1043.865,147.257,-92.848,170.496,37.947,157.152
C07781=1043.871,147.505,-92.871,170.498,37.949,157.152
C07782=1043.878,147.755,-92.892,170.499,37.950,157.153
C07783=1043.884,148.004,-92.914,170.502,37.951,157.153
C07784=1043.890,148.253,-92.936,170.504,37.952,157.153
C07785=1043.896,148.502,-92.958,170.506,37.953,157.153
C07786=1043.903,148.751,-92.980,170.508,37.955,157.154
C07787=1043.909,149.000,-93.001,170.511,37.956,157.154
C07788=1043.914,149.249,-93.023,170.513,37.957,157.154
C07789=1043.920,149.497,-93.045,170.515,37.959,157.155
C07790=1043.926,149.747,-93.067,170.517,37.960,157.155
C07791=1043.933,149.995,-93.089,170.519,37.962,157.155
C07792=1043.939,150.244,-93.111,170.522,37.963,157.155
C07793=1043.945,150.494,-93.133,170.524,37.964,157.156
C07794=1043.951,150.742,-93.156,170.526,37.966,157.156
C07795=1043.957,150.992,-93.177,170.528,37.967,157.156
C07796=1043.963,151.241,-93.199,170.531,37.968,157.157
C07797=1043.969,151.489,-93.221,170.533,37.969,157.157
C07798=1043.975,151.738,-93.242,170.535,37.971,157.157
C07799=1043.981,151.987,-93.265,170.537,37.972,157.158
C07800=1043.987,152.236,-93.287,170.540,37.973,157.158
C07801=1043.993,152.485,-93.309,170.542,37.974,157.158
C07802=1044.000,152.734,-93.331,170.544,37.976,157.158
C07803=1044.005,152.983,-93.353,170.546,37.977,157.159
C07804=1044.012,153.232,-93.376,170.549,37.979,157.159
C07805=1044.018,153.481,-93.397,170.551,37.980,157.159
C07806=1044.024,153.730,-93.420,170.553,37.981,157.160
C07807=1044.030,153.979,-93.441,170.554,37.983,157.160
C07808=1044.036,154.228,-93.464,170.556,37.984,157.160
C07809=1044.042,154.477,-93.486,170.559,37.985,157.160
C07810=1044.049,154.726,-93.508,170.561,37.987,157.161
C07811=1044.054,154.975,-93.530,170.563,37.988,157.161
C07812=1044.061,155.224,-93.553,170.565,37.989,157.161
C07813=1044.067,155.472,-93.575,170.568,37.991,157.162
C07814=1044.072,155.722,-93.597,170.570,37.992,157.162
C07815=1044.079,155.970,-93.620,170.572,37.993,157.162
C07816=1044.085,156.219,-93.641,170.574,37.995,157.163
C07817=1044.090,156.468,-93.664,170.577,37.996,157.163
C07818=1044.097,156.716,-93.686,170.579,37.997,157.163
C07819=1044.102,156.966,-93.708,170.581,37.999,157.164
C07820=1044.110,157.251,-93.735,170.584,38.000,157.164
C07821=1044.117,157.537,-93.760,170.587,38.002,157.164
C07822=1044.124,157.821,-93.786,170.589,38.004,157.165
C07823=1044.131,158.107,-93.811,170.592,38.005,157.165
C07824=1044.137,158.356,-93.834,170.595,38.007,157.165
C07825=1044.143,158.605,-93.855,170.597,38.008,157.166
C07826=1044.149,158.854,-93.878,170.599,38.009,157.166
C07827=1044.155,159.103,-93.901,170.601,38.011,157.166
C07828=1044.161,159.352,-93.922,170.604,38.012,157.167
C07829=1044.168,159.601,-93.945,170.606,38.013,157.167
C07830=1044.173,159.849,-93.968,170.608,38.015,157.167
C07831=1044.180,160.098,-93.990,170.610,38.016,157.167
C07832=1044.185,160.348,-94.012,170.612,38.017,157.168
C07833=1044.192,160.596,-94.035,170.615,38.019,157.168
C07834=1044.198,160.846,-94.058,170.617,38.020,157.168
C07835=1044.204,161.095,-94.081,170.619,38.022,157.169
C07836=1044.209,161.343,-94.104,170.622,38.023,157.169
C07837=1044.215,161.592,-94.127,170.624,38.025,157.169
C07838=1044.222,161.841,-94.149,170.626,38.027,157.170
C07839=1044.227,162.090,-94.171,170.628,38.028,157.170
C07840=1044.233,162.339,-94.194,170.631,38.030,157.171
C07841=1044.239,162.588,-94.217,170.633,38.031,157.171
C07842=1044.245,162.837,-94.240,170.635,38.033,157.171
C07843=1044.251,163.086,-94.263,170.637,38.034,157.171
C07844=1044.256,163.335,-94.285,170.640,38.036,157.172
C07845=1044.262,163.584,-94.308,170.642,38.037,157.172
C07846=1044.268,163.832,-94.331,170.644,38.038,157.173
C07847=1044.274,164.081,-94.354,170.647,38.040,157.173
C07848=1044.280,164.330,-94.377,170.649,38.041,157.173
C07849=1044.286,164.579,-94.400,170.651,38.043,157.174
C07850=1044.292,164.828,-94.423,170.653,38.044,157.174
C07851=1044.297,165.077,-94.446,170.656,38.046,157.174
C07852=1044.304,165.325,-94.468,170.658,38.047,157.175
C07853=1044.310,165.574,-94.491,170.660,38.049,157.175
C07854=1044.315,165.823,-94.514,170.662,38.050,157.175
C07855=1044.321,166.072,-94.537,170.665,38.052,157.176
C07856=1044.327,166.322,-94.560,170.667,38.054,157.176
C07857=1044.334,166.570,-94.582,170.669,38.055,157.176
C07858=1044.340,166.819,-94.605,170.672,38.057,157.177
C07859=1044.345,167.068,-94.628,170.674,38.058,157.177
C07860=1044.351,167.317,-94.651,170.676,38.060,157.177
C07861=1044.357,167.565,-94.675,170.678,38.061,157.178
C07862=1044.363,167.814,-94.698,170.682,38.063,157.178
C07863=1044.369,168.063,-94.720,170.684,38.064,157.178
C07864=1044.376,168.312,-94.743,170.686,38.065,157.179
C07865=1044.381,168.561,-94.766,170.689,38.067,157.179
C07866=1044.387,168.810,-94.789,170.691,38.068,157.179
C07867=1044.393,169.059,-94.812,170.693,38.070,157.180
C07868=1044.400,169.307,-94.835,170.695,38.071,157.180
C07869=1044.405,169.556,-94.858,170.698,38.073,157.180
C07870=1044.412,169.805,-94.882,170.700,38.074,157.181
C07871=1044.417,170.054,-94.905,170.702,38.076,157.181
C07872=1044.423,170.303,-94.928,170.704,38.078,157.181
C07873=1044.429,170.551,-94.951,170.707,38.079,157.182
C07874=1044.435,170.800,-94.974,170.709,38.081,157.182
C07875=1044.442,171.050,-94.997,170.712,38.082,157.182
C07876=1044.448,171.298,-95.020,170.715,38.084,157.183
C07877=1044.453,171.547,-95.043,170.717,38.085,157.183
C07878=1044.459,171.796,-95.066,170.719,38.087,157.183
C07879=1044.466,172.045,-95.090,170.721,38.088,157.184
C07880=1044.471,172.294,-95.113,170.724,38.089,157.184
C07881=1044.478,172.542,-95.136,170.726,38.091,157.184
C07882=1044.484,172.791,-95.159,170.728,38.092,157.185
C07883=1044.490,173.041,-95.182,170.730,38.094,157.185
C07884=1044.497,173.325,-95.209,170.734,38.096,157.186
C07885=1044.504,173.610,-95.235,170.736,38.098,157.186
C07886=1044.511,173.895,-95.262,170.739,38.099,157.186
C07887=1044.517,174.179,-95.289,170.742,38.101,157.187
C07888=1044.524,174.429,-95.311,170.744,38.102,157.187
C07889=1044.531,174.677,-95.335,170.746,38.104,157.187
C07890=1044.536,174.926,-95.358,170.750,38.106,157.188
C07891=1044.542,175.175,-95.381,170.752,38.107,157.188
C07892=1044.549,175.424,-95.405,170.754,38.109,157.188
C07893=1044.554,175.673,-95.428,170.756,38.110,157.189
C07894=1044.560,175.921,-95.452,170.759,38.112,157.189
C07895=1044.567,176.171,-95.475,170.761,38.113,157.190
C07896=1044.573,176.419,-95.497,170.764,38.115,157.190
C07897=1044.579,176.667,-95.521,170.767,38.116,157.190
C07898=1044.586,176.917,-95.544,170.769,38.117,157.190
C07899=1044.592,177.165,-95.568,170.771,38.119,157.191
C07900=1044.598,177.415,-95.591,170.773,38.121,157.191
C07901=1044.604,177.663,-95.615,170.776,38.122,157.192
C07902=1044.610,177.912,-95.638,170.779,38.124,157.192
C07903=1044.616,178.161,-95.662,170.781,38.125,157.192
C07904=1044.622,178.410,-95.685,170.784,38.127,157.193
C07905=1044.629,178.659,-95.709,170.786,38.129,157.193
C07906=1044.634,178.908,-95.732,170.788,38.130,157.193
C07907=1044.641,179.156,-95.755,170.790,38.131,157.194
C07908=1044.648,179.405,-95.779,170.794,38.133,157.194
C07909=1044.654,179.654,-95.802,170.796,38.134,157.194
C07910=1044.660,179.903,-95.826,170.798,38.136,157.195
C07911=1044.666,180.152,-95.849,170.801,38.137,157.195
C07912=1044.673,180.401,-95.873,170.803,38.139,157.195
C07913=1044.678,180.649,-95.896,170.806,38.141,157.196
C07914=1044.684,180.898,-95.919,170.808,38.142,157.196
C07915=1044.691,181.147,-95.943,170.811,38.144,157.196
C07916=1044.697,181.396,-95.966,170.813,38.145,157.197
C07917=1044.703,181.645,-95.990,170.816,38.147,157.197
C07918=1044.709,181.893,-96.014,170.819,38.148,157.198
C07919=1044.716,182.142,-96.037,170.821,38.150,157.198
C07920=1044.723,182.390,-96.060,170.823,38.151,157.198
C07921=1044.729,182.639,-96.084,170.825,38.153,157.199
C07922=1044.735,182.888,-96.107,170.829,38.155,157.199
C07923=1044.742,183.137,-96.131,170.831,38.156,157.199
C07924=1044.748,183.386,-96.155,170.833,38.158,157.200
C07925=1044.754,183.635,-96.178,170.836,38.159,157.200
C07926=1044.760,183.883,-96.202,170.839,38.160,157.200
C07927=1044.766,184.133,-96.227,170.841,38.162,157.201
C07928=1044.772,184.381,-96.250,170.844,38.164,157.201
C07929=1044.778,184.630,-96.275,170.846,38.166,157.202
C07930=1044.784,184.879,-96.299,170.848,38.167,157.202
C07931=1044.789,185.127,-96.323,170.852,38.169,157.202
C07932=1044.796,185.376,-96.347,170.854,38.171,157.203
C07933=1044.801,185.625,-96.370,170.856,38.173,157.203
C07934=1044.807,185.874,-96.394,170.859,38.174,157.204
C07935=1044.813,186.123,-96.419,170.861,38.176,157.204
C07936=1044.819,186.372,-96.443,170.864,38.178,157.204
C07937=1044.825,186.620,-96.467,170.867,38.180,157.205
C07938=1044.831,186.869,-96.491,170.869,38.181,157.205
C07939=1044.837,187.118,-96.515,170.871,38.183,157.206
C07940=1044.843,187.366,-96.539,170.874,38.185,157.206
C07941=1044.848,187.616,-96.564,170.877,38.187,157.206
C07942=1044.855,187.864,-96.587,170.879,38.188,157.207
C07943=1044.860,188.113,-96.612,170.882,38.190,157.207
C07944=1044.866,188.361,-96.636,170.884,38.192,157.208
C07945=1044.873,188.610,-96.660,170.887,38.194,157.208
C07946=1044.879,188.858,-96.685,170.890,38.195,157.208
C07947=1044.885,189.108,-96.709,170.892,38.197,157.209
C07948=1044.892,189.393,-96.736,170.895,38.199,157.209
C07949=1044.898,189.677,-96.763,170.898,38.201,157.210
C07950=1044.905,189.961,-96.792,170.901,38.203,157.210
C07951=1044.913,190.246,-96.819,170.903,38.205,157.211
C07952=1044.918,190.494,-96.844,170.907,38.206,157.211
C07953=1044.925,190.743,-96.868,170.909,38.208,157.211
C07954=1044.931,190.992,-96.893,170.911,38.210,157.212
C07955=1044.937,191.240,-96.916,170.914,38.212,157.212
C07956=1044.943,191.490,-96.941,170.917,38.213,157.213
C07957=1044.949,191.738,-96.964,170.919,38.215,157.213
C07958=1044.955,191.986,-96.990,170.922,38.218,157.213
C07959=1044.961,192.236,-97.014,170.925,38.219,157.214
C07960=1044.967,192.484,-97.038,170.927,38.221,157.214
C07961=1044.973,192.733,-97.063,170.930,38.223,157.215
C07962=1044.979,192.982,-97.086,170.932,38.225,157.215
C07963=1044.985,193.230,-97.112,170.935,38.226,157.216
C07964=1044.992,193.479,-97.136,170.938,38.228,157.216
C07965=1044.997,193.728,-97.160,170.940,38.230,157.216
C07966=1045.003,193.977,-97.184,170.943,38.232,157.217
C07967=1045.010,194.225,-97.209,170.946,38.233,157.217
C07968=1045.016,194.474,-97.233,170.948,38.235,157.218
C07969=1045.022,194.723,-97.258,170.951,38.237,157.218
C07970=1045.028,194.972,-97.283,170.954,38.238,157.218
C07971=1045.034,195.220,-97.307,170.956,38.240,157.219
C07972=1045.040,195.469,-97.331,170.958,38.242,157.219
C07973=1045.047,195.718,-97.356,170.962,38.244,157.220
C07974=1045.052,195.966,-97.380,170.964,38.245,157.220
C07975=1045.059,196.215,-97.404,170.966,38.247,157.220
C07976=1045.065,196.464,-97.430,170.970,38.250,157.221
C07977=1045.071,196.713,-97.454,170.972,38.251,157.221
C07978=1045.077,196.961,-97.479,170.975,38.253,157.222
C07979=1045.083,197.210,-97.503,170.978,38.255,157.222
C07980=1045.090,197.459,-97.527,170.980,38.256,157.222
C07981=1045.095,197.707,-97.552,170.984,38.258,157.223
C07982=1045.102,197.956,-97.576,170.986,38.260,157.223
C07983=1045.108,198.205,-97.602,170.988,38.262,157.224
C07984=1045.115,198.454,-97.626,170.992,38.263,157.224
C07985=1045.121,198.702,-97.651,170.994,38.265,157.225
C07986=1045.126,198.951,-97.675,170.996,38.267,157.225
C07987=1045.133,199.199,-97.700,171.000,38.269,157.225
C07988=1045.139,199.449,-97.725,171.002,38.271,157.226
C07989=1045.146,199.697,-97.749,171.004,38.273,157.226
C07990=1045.151,199.946,-97.774,171.008,38.274,157.227
C07991=1045.158,200.194,-97.799,171.010,38.276,157.227
C07992=1045.164,200.443,-97.823,171.013,38.278,157.227
C07993=1045.170,200.692,-97.848,171.016,38.280,157.228
C07994=1045.177,200.940,-97.873,171.018,38.282,157.228
C07995=1045.183,201.190,-97.898,171.021,38.284,157.229
C07996=1045.189,201.437,-97.923,171.024,38.285,157.229
C07997=1045.195,201.687,-97.947,171.027,38.287,157.230
C07998=1045.201,201.935,-97.973,171.030,38.289,157.230
C07999=1045.207,202.184,-97.998,171.032,38.291,157.231
C08000=1045.213,202.433,-98.023,171.035,38.293,157.231
C08001=1045.219,202.681,-98.047,171.038,38.295,157.232
C08002=1045.226,202.930,-98.072,171.040,38.297,157.232
C08003=1045.232,203.178,-98.098,171.043,38.299,157.232
C08004=1045.238,203.428,-98.122,171.046,38.301,157.233
C08005=1045.244,203.676,-98.148,171.049,38.303,157.233
C08006=1045.250,203.925,-98.173,171.052,38.304,157.234
C08007=1045.256,204.173,-98.198,171.054,38.307,157.234
C08008=1045.262,204.422,-98.223,171.057,38.309,157.235
C08009=1045.268,204.671,-98.248,171.060,38.310,157.235
C08010=1045.274,204.920,-98.273,171.063,38.313,157.236
C08011=1045.280,205.168,-98.299,171.065,38.314,157.236
C08012=1045.306,206.220,-98.405,171.323,38.415,157.262
C08013=1045.313,206.498,-98.434,171.326,38.418,157.263
C08014=1045.321,206.775,-98.463,171.327,38.421,157.264
C08015=1045.329,207.055,-98.492,171.330,38.424,157.264
C08016=1045.336,207.333,-98.522,171.332,38.427,157.265
C08017=1045.343,207.581,-98.548,171.334,38.430,157.265
C08018=1045.349,207.830,-98.575,171.336,38.433,157.266
C08019=1045.356,208.078,-98.601,171.339,38.435,157.267
C08020=1045.363,208.327,-98.628,171.340,38.438,157.267
C08021=1045.368,208.575,-98.654,171.343,38.441,157.268
C08022=1045.376,208.824,-98.681,171.345,38.443,157.268
C08023=1045.382,209.072,-98.707,171.347,38.446,157.269
C08024=1045.388,209.321,-98.734,171.349,38.449,157.270
C08025=1045.395,209.569,-98.760,171.351,38.451,157.270
C08026=1045.402,209.818,-98.786,171.353,38.454,157.271
C08027=1045.408,210.066,-98.813,171.355,38.457,157.271
C08028=1045.415,210.315,-98.839,171.358,38.460,157.272
C08029=1045.421,210.563,-98.865,171.359,38.463,157.273
C08030=1045.428,210.812,-98.892,171.362,38.465,157.273
C08031=1045.434,211.060,-98.918,171.363,38.468,157.274
C08032=1045.441,211.309,-98.945,171.366,38.470,157.275
C08033=1045.447,211.557,-98.971,171.368,38.473,157.275
C08034=1045.454,211.806,-98.998,171.370,38.476,157.276
C08035=1045.460,212.054,-99.025,171.372,38.479,157.276
C08036=1045.467,212.303,-99.051,171.374,38.482,157.277
C08037=1045.473,212.551,-99.078,171.376,38.484,157.278
C08038=1045.479,212.800,-99.105,171.379,38.487,157.278
C08039=1045.487,213.048,-99.132,171.381,38.490,157.279
C08040=1045.493,213.297,-99.158,171.383,38.492,157.279
C08041=1045.500,213.546,-99.185,171.385,38.495,157.280
C08042=1045.505,213.794,-99.211,171.387,38.498,157.281
C08043=1045.513,214.043,-99.238,171.390,38.500,157.281
C08044=1045.519,214.290,-99.265,171.391,38.503,157.282
C08045=1045.526,214.539,-99.292,171.394,38.506,157.283
C08046=1045.532,214.787,-99.318,171.395,38.509,157.283
C08047=1045.538,215.037,-99.345,171.398,38.511,157.284
C08048=1045.545,215.285,-99.372,171.400,38.514,157.284
C08049=1045.551,215.533,-99.399,171.402,38.517,157.285
C08050=1045.558,215.782,-99.426,171.404,38.519,157.286
C08051=1045.564,216.030,-99.452,171.407,38.522,157.286
C08052=1045.571,216.279,-99.479,171.408,38.525,157.287
C08053=1045.578,216.527,-99.506,171.411,38.528,157.287
C08054=1045.584,216.776,-99.533,171.414,38.530,157.288
C08055=1045.591,217.024,-99.559,171.415,38.533,157.289
C08056=1045.597,217.273,-99.587,171.418,38.536,157.289
C08057=1045.604,217.521,-99.613,171.420,38.538,157.290
C08058=1045.610,217.770,-99.640,171.422,38.541,157.291
C08059=1045.616,218.018,-99.668,171.424,38.543,157.291
C08060=1045.623,218.266,-99.694,171.427,38.546,157.292
C08061=1045.630,218.516,-99.721,171.428,38.549,157.292
C08062=1045.637,218.763,-99.748,171.431,38.552,157.293
C08063=1045.643,219.012,-99.775,171.433,38.554,157.294
C08064=1045.650,219.260,-99.802,171.435,38.557,157.294
C08065=1045.657,219.509,-99.829,171.437,38.559,157.295
C08066=1045.663,219.758,-99.856,171.440,38.562,157.295
C08067=1045.670,220.006,-99.883,171.441,38.565,157.296
C08068=1045.676,220.255,-99.910,171.444,38.568,157.297
C08069=1045.684,220.537,-99.941,171.447,38.570,157.297
C08070=1045.691,220.822,-99.972,171.449,38.573,157.298
C08071=1045.698,221.105,-100.003,171.452,38.577,157.299
C08072=1045.706,221.389,-100.033,171.455,38.580,157.299
C08073=1045.712,221.637,-100.061,171.457,38.582,157.300
C08074=1045.719,221.886,-100.088,171.459,38.585,157.301
C08075=1045.725,222.135,-100.116,171.461,38.588,157.301
C08076=1045.731,222.383,-100.143,171.464,38.590,157.302
C08077=1045.739,222.631,-100.170,171.465,38.593,157.302
C08078=1045.745,222.880,-100.197,171.468,38.596,157.303
C08079=1045.751,223.128,-100.224,171.470,38.599,157.304
C08080=1045.758,223.376,-100.252,171.473,38.602,157.304
C08081=1045.764,223.625,-100.279,171.474,38.604,157.305
C08082=1045.771,223.874,-100.307,171.477,38.607,157.306
C08083=1045.777,224.122,-100.334,171.479,38.609,157.306
C08084=1045.784,224.370,-100.360,171.481,38.612,157.307
C08085=1045.791,224.619,-100.388,171.483,38.614,157.307
C08086=1045.797,224.867,-100.416,171.486,38.617,157.308
C08087=1045.803,225.116,-100.442,171.489,38.620,157.309
C08088=1045.810,225.364,-100.470,171.490,38.623,157.309
C08089=1045.816,225.613,-100.498,171.493,38.626,157.310
C08090=1045.823,225.861,-100.526,171.495,38.628,157.310
C08091=1045.829,226.109,-100.552,171.498,38.631,157.311
C08092=1045.836,226.357,-100.579,171.500,38.633,157.312
C08093=1045.843,226.606,-100.607,171.502,38.636,157.312
C08094=1045.850,226.854,-100.635,171.504,38.638,157.313
C08095=1045.856,227.103,-100.662,171.507,38.641,157.314
C08096=1045.862,227.351,-100.689,171.509,38.644,157.314
C08097=1045.869,227.600,-100.717,171.511,38.647,157.315
C08098=1045.876,227.848,-100.745,171.514,38.649,157.315
C08099=1045.882,228.097,-100.772,171.516,38.652,157.316
C08100=1045.889,228.346,-100.800,171.519,38.654,157.317
C08101=1045.895,228.594,-100.827,171.521,38.657,157.317
C08102=1045.902,228.842,-100.855,171.523,38.659,157.318
C08103=1045.908,229.090,-100.882,171.525,38.662,157.318
C08104=1045.915,229.339,-100.910,171.528,38.665,157.319
C08105=1045.921,229.587,-100.938,171.530,38.668,157.320
C08106=1045.928,229.835,-100.966,171.533,38.671,157.320
C08107=1045.935,230.084,-100.993,171.534,38.673,157.321
C08108=1045.941,230.332,-101.021,171.537,38.676,157.322
C08109=1045.947,230.581,-101.048,171.540,38.678,157.322
C08110=1045.954,230.829,-101.075,171.542,38.681,157.323
C08111=1045.960,231.078,-101.104,171.545,38.684,157.323
C08112=1045.967,231.326,-101.131,171.546,38.686,157.324
C08113=1045.973,231.575,-101.159,171.549,38.689,157.325
C08114=1045.980,231.823,-101.187,171.551,38.692,157.325
C08115=1045.987,232.072,-101.215,171.554,38.694,157.326
C08116=1045.993,232.319,-101.242,171.556,38.697,157.326
C08117=1046.000,232.567,-101.270,171.559,38.700,157.327
C08118=1046.006,232.816,-101.299,171.561,38.703,157.328
C08119=1046.012,233.064,-101.326,171.563,38.705,157.328
C08120=1046.019,233.313,-101.354,171.566,38.708,157.329
C08121=1046.026,233.561,-101.382,171.568,38.710,157.330
C08122=1046.032,233.810,-101.410,171.571,38.713,157.330
C08123=1046.038,234.058,-101.438,171.573,38.716,157.331
C08124=1046.045,234.307,-101.466,171.575,38.718,157.331
C08125=1046.052,234.583,-101.498,171.578,38.721,157.332
C08126=1046.059,234.859,-101.528,171.581,38.724,157.333
C08127=1046.067,235.135,-101.559,171.584,38.727,157.333
C08128=1046.073,235.411,-101.591,171.586,38.731,157.334
C08129=1046.080,235.660,-101.618,171.589,38.733,157.335
C08130=1046.087,235.908,-101.647,171.591,38.736,157.336
C08131=1046.093,236.156,-101.675,171.593,38.738,157.336
C08132=1046.100,236.405,-101.703,171.596,38.741,157.337
C08133=1046.106,236.653,-101.731,171.598,38.743,157.337
C08134=1046.113,236.902,-101.758,171.601,38.746,157.338
C08135=1046.119,237.150,-101.787,171.603,38.749,157.339
C08136=1046.126,237.398,-101.815,171.606,38.751,157.339
C08137=1046.133,237.647,-101.843,171.608,38.754,157.340
C08138=1046.139,237.895,-101.872,171.611,38.757,157.340
C08139=1046.146,238.143,-101.900,171.614,38.760,157.341
C08140=1046.152,238.392,-101.927,171.615,38.762,157.342
C08141=1046.159,238.640,-101.956,171.618,38.765,157.342
C08142=1046.165,238.888,-101.984,171.620,38.767,157.343
C08143=1046.172,239.137,-102.012,171.623,38.770,157.344
C08144=1046.178,239.385,-102.041,171.625,38.772,157.344
C08145=1046.185,239.633,-102.069,171.628,38.775,157.345
C08146=1046.192,239.881,-102.097,171.630,38.778,157.345
C08147=1046.198,240.130,-102.125,171.633,38.780,157.346
C08148=1046.204,240.378,-102.153,171.636,38.783,157.347
C08149=1046.211,240.627,-102.182,171.638,38.786,157.347
C08150=1046.217,240.875,-102.210,171.641,38.788,157.348
C08151=1046.224,241.123,-102.238,171.643,38.791,157.349
C08152=1046.230,241.372,-102.267,171.646,38.794,157.349
C08153=1046.237,241.619,-102.295,171.648,38.796,157.350
C08154=1046.243,241.868,-102.323,171.650,38.799,157.350
C08155=1046.250,242.116,-102.352,171.653,38.802,157.351
C08156=1046.256,242.365,-102.380,171.655,38.804,157.352
C08157=1046.262,242.613,-102.409,171.658,38.807,157.352
C08158=1046.269,242.861,-102.438,171.660,38.810,157.353
C08159=1046.275,243.109,-102.466,171.663,38.812,157.354
C08160=1046.282,243.357,-102.494,171.665,38.815,157.354
C08161=1046.289,243.607,-102.523,171.668,38.818,157.355
C08162=1046.295,243.855,-102.552,171.670,38.820,157.355
C08163=1046.302,244.103,-102.581,171.673,38.823,157.356
C08164=1046.308,244.351,-102.609,171.676,38.825,157.357
C08165=1046.315,244.599,-102.637,171.678,38.828,157.357
C08166=1046.321,244.847,-102.666,171.681,38.831,157.358
C08167=1046.327,245.096,-102.695,171.683,38.834,157.359
C08168=1046.334,245.344,-102.723,171.686,38.836,157.359
C08169=1046.340,245.592,-102.752,171.689,38.839,157.360
C08170=1046.346,245.841,-102.781,171.691,38.842,157.361
C08171=1046.353,246.089,-102.810,171.694,38.845,157.361
C08172=1046.360,246.337,-102.838,171.696,38.847,157.362
C08173=1046.366,246.586,-102.867,171.699,38.850,157.362
C08174=1046.373,246.834,-102.896,171.701,38.853,157.363
C08175=1046.379,247.082,-102.925,171.704,38.855,157.364
C08176=1046.385,247.331,-102.954,171.707,38.858,157.365
C08177=1046.391,247.579,-102.983,171.709,38.861,157.365
C08178=1046.397,247.827,-103.012,171.712,38.864,157.366
C08179=1046.404,248.075,-103.040,171.714,38.866,157.366
C08180=1046.411,248.323,-103.069,171.717,38.869,157.367
C08181=1046.418,248.594,-103.101,171.720,38.872,157.368
C08182=1046.425,248.864,-103.133,171.722,38.875,157.369
C08183=1046.432,249.134,-103.164,171.725,38.878,157.369
C08184=1046.439,249.405,-103.196,171.729,38.881,157.370
C08185=1046.445,249.653,-103.225,171.731,38.884,157.371
C08186=1046.452,249.902,-103.254,171.734,38.886,157.371
C08187=1046.458,250.150,-103.283,171.736,38.889,157.372
C08188=1046.464,250.398,-103.312,171.739,38.892,157.373
C08189=1046.470,250.646,-103.341,171.741,38.894,157.373
C08190=1046.477,250.894,-103.370,171.744,38.897,157.374
C08191=1046.484,251.143,-103.399,171.747,38.900,157.374
C08192=1046.491,251.391,-103.428,171.749,38.902,157.375
C08193=1046.497,251.639,-103.457,171.752,38.905,157.376
C08194=1046.503,251.887,-103.486,171.754,38.908,157.376
C08195=1046.509,252.135,-103.515,171.757,38.910,157.377
C08196=1046.516,252.384,-103.545,171.760,38.913,157.378
C08197=1046.522,252.632,-103.574,171.762,38.916,157.378
C08198=1046.529,252.880,-103.603,171.765,38.918,157.379
C08199=1046.535,253.128,-103.632,171.767,38.921,157.380
C08200=1046.543,253.376,-103.661,171.770,38.924,157.380
C08201=1046.549,253.624,-103.690,171.774,38.926,157.381
C08202=1046.555,253.873,-103.719,171.776,38.929,157.382
C08203=1046.562,254.121,-103.749,171.779,38.932,157.382
C08204=1046.568,254.370,-103.778,171.781,38.934,157.383
C08205=1046.575,254.618,-103.807,171.784,38.937,157.383
C08206=1046.581,254.865,-103.837,171.787,38.940,157.384
C08207=1046.588,255.114,-103.866,171.789,38.942,157.385
C08208=1046.594,255.362,-103.895,171.792,38.945,157.385
C08209=1046.601,255.610,-103.924,171.794,38.948,157.386
C08210=1046.607,255.859,-103.953,171.798,38.950,157.387
C08211=1046.614,256.107,-103.983,171.801,38.953,157.387
C08212=1046.621,256.356,-104.013,171.803,38.956,157.388
C08213=1046.628,256.603,-104.041,171.806,38.958,157.389
C08214=1046.634,256.851,-104.071,171.808,38.961,157.389
C08215=1046.641,257.100,-104.100,171.811,38.964,157.390
C08216=1046.647,257.348,-104.129,171.813,38.966,157.391
C08217=1046.654,257.596,-104.158,171.817,38.969,157.391
C08218=1046.661,257.844,-104.188,171.820,38.972,157.392
C08219=1046.667,258.092,-104.217,171.822,38.974,157.392
C08220=1046.674,258.341,-104.247,171.825,38.977,157.393
C08221=1046.680,258.589,-104.277,171.827,38.980,157.394
C08222=1046.687,258.837,-104.306,171.830,38.982,157.394
C08223=1046.694,259.085,-104.336,171.834,38.985,157.395
C08224=1046.700,259.333,-104.365,171.836,38.987,157.396
C08225=1046.707,259.582,-104.394,171.839,38.990,157.396
C08226=1046.714,259.829,-104.424,171.841,38.993,157.397
C08227=1046.720,260.078,-104.453,171.844,38.995,157.398
C08228=1046.727,260.326,-104.483,171.848,38.998,157.398
C08229=1046.734,260.575,-104.513,171.850,39.001,157.399
C08230=1046.740,260.822,-104.542,171.853,39.003,157.400
C08231=1046.747,261.071,-104.572,171.855,39.006,157.400
C08232=1046.754,261.318,-104.601,171.858,39.009,157.401
C08233=1046.761,261.567,-104.631,171.862,39.011,157.402
C08234=1046.767,261.815,-104.661,171.864,39.014,157.402
C08235=1046.774,262.064,-104.690,171.867,39.016,157.403
C08236=1046.781,262.311,-104.720,171.869,39.019,157.403
C08237=1046.788,262.581,-104.751,171.873,39.022,157.404
C08238=1046.795,262.849,-104.784,171.876,39.025,157.405
C08239=1046.802,263.118,-104.816,171.878,39.028,157.406
C08240=1046.809,263.387,-104.849,171.882,39.031,157.406
C08241=1046.816,263.634,-104.878,171.885,39.034,157.407
C08242=1046.822,263.883,-104.909,171.887,39.036,157.408
C08243=1046.828,264.131,-104.938,171.890,39.039,157.408
C08244=1046.836,264.379,-104.968,171.894,39.042,157.409
C08245=1046.841,264.627,-104.999,171.896,39.045,157.410
C08246=1046.848,264.876,-105.028,171.899,39.048,157.410
C08247=1046.854,265.124,-105.058,171.901,39.050,157.411
C08248=1046.861,265.372,-105.088,171.905,39.053,157.412
C08249=1046.868,265.619,-105.118,171.908,39.056,157.412
C08250=1046.874,265.868,-105.149,171.910,39.058,157.413
C08251=1046.881,266.116,-105.178,171.913,39.061,157.414
C08252=1046.888,266.364,-105.208,171.916,39.064,157.414
C08253=1046.893,266.612,-105.238,171.919,39.066,157.415
C08254=1046.901,266.860,-105.268,171.922,39.069,157.416
C08255=1046.907,267.108,-105.298,171.924,39.072,157.416
C08256=1046.914,267.356,-105.329,171.928,39.075,157.417
C08257=1046.921,267.605,-105.359,171.931,39.077,157.418
C08258=1046.927,267.852,-105.389,171.933,39.080,157.418
C08259=1046.933,268.101,-105.419,171.937,39.083,157.419
C08260=1046.940,268.349,-105.449,171.940,39.086,157.420
C08261=1046.946,268.597,-105.479,171.942,39.089,157.421
C08262=1046.953,268.845,-105.509,171.945,39.091,157.421
C08263=1046.959,269.093,-105.540,171.948,39.094,157.422
C08264=1046.967,269.341,-105.570,171.951,39.096,157.423
C08265=1046.972,269.589,-105.600,171.954,39.099,157.423
C08266=1046.980,269.838,-105.630,171.957,39.102,157.424
C08267=1046.986,270.085,-105.661,171.960,39.105,157.425
C08268=1046.993,270.333,-105.692,171.963,39.108,157.425
C08269=1046.999,270.581,-105.722,171.965,39.111,157.426
C08270=1047.006,270.829,-105.752,171.969,39.113,157.427
C08271=1047.012,271.077,-105.783,171.971,39.116,157.427
C08272=1047.019,271.326,-105.813,171.974,39.119,157.428
C08273=1047.025,271.574,-105.843,171.978,39.121,157.429
C08274=1047.032,271.822,-105.874,171.980,39.124,157.429
C08275=1047.039,272.070,-105.904,171.983,39.127,157.430
C08276=1047.045,272.317,-105.935,171.987,39.130,157.431
C08277=1047.052,272.566,-105.965,171.989,39.133,157.432
C08278=1047.058,272.813,-105.996,171.992,39.135,157.432
C08279=1047.064,273.062,-106.026,171.996,39.138,157.433
C08280=1047.072,273.310,-106.057,171.998,39.141,157.434
C08281=1047.078,273.557,-106.088,172.001,39.143,157.434
C08282=1047.084,273.806,-106.118,172.005,39.146,157.435
C08283=1047.091,274.054,-106.148,172.007,39.149,157.436
C08284=1047.098,274.302,-106.180,172.010,39.152,157.436
C08285=1047.104,274.550,-106.210,172.014,39.155,157.437
C08286=1047.110,274.798,-106.241,172.016,39.157,157.438
C08287=1047.118,275.046,-106.272,172.019,39.160,157.438
C08288=1047.123,275.294,-106.302,172.023,39.163,157.439
C08289=1047.130,275.542,-106.333,172.025,39.166,157.440
C08290=1047.137,275.790,-106.364,172.029,39.169,157.441
C08291=1047.144,276.038,-106.394,172.032,39.172,157.441
C08292=1047.150,276.286,-106.425,172.034,39.174,157.442
C08293=1047.158,276.559,-106.459,172.038,39.177,157.443
C08294=1047.165,276.832,-106.493,172.042,39.181,157.443
C08295=1047.172,277.106,-106.527,172.044,39.183,157.444
C08296=1047.179,277.379,-106.561,172.048,39.187,157.445
C08297=1047.185,277.627,-106.591,172.051,39.190,157.446
C08298=1047.192,277.875,-106.623,172.054,39.192,157.446
C08299=1047.199,278.124,-106.654,172.057,39.195,157.447
C08300=1047.205,278.371,-106.685,172.061,39.198,157.448
C08301=1047.212,278.619,-106.715,172.063,39.201,157.449
C08302=1047.219,278.867,-106.746,172.066,39.204,157.449
C08303=1047.225,279.115,-106.778,172.070,39.206,157.450
C08304=1047.232,279.363,-106.808,172.072,39.209,157.451
C08305=1047.238,279.611,-106.840,172.076,39.212,157.451
C08306=1047.245,279.858,-106.871,172.079,39.215,157.452
C08307=1047.251,280.107,-106.902,172.081,39.218,157.453
C08308=1047.258,280.355,-106.933,172.085,39.220,157.454
C08309=1047.264,280.603,-106.964,172.088,39.223,157.454
C08310=1047.271,280.851,-106.995,172.092,39.227,157.455
C08311=1047.277,281.098,-107.026,172.094,39.230,157.456
C08312=1047.284,281.346,-107.058,172.098,39.232,157.457
C08313=1047.290,281.594,-107.089,172.101,39.235,157.457
C08314=1047.297,281.843,-107.120,172.104,39.238,157.458
C08315=1047.304,282.091,-107.151,172.107,39.241,157.459
C08316=1047.310,282.339,-107.183,172.110,39.244,157.459
C08317=1047.316,282.586,-107.214,172.113,39.246,157.460
C08318=1047.323,282.834,-107.245,172.116,39.249,157.461
C08319=1047.330,283.082,-107.276,172.120,39.252,157.461
C08320=1047.336,283.330,-107.307,172.122,39.255,157.462
C08321=1047.343,283.578,-107.339,172.126,39.258,157.463
C08322=1047.350,283.826,-107.370,172.129,39.261,157.464
C08323=1047.356,284.074,-107.402,172.133,39.264,157.464
C08324=1047.363,284.322,-107.433,172.135,39.267,157.465
C08325=1047.370,284.570,-107.464,172.139,39.269,157.466
C08326=1047.377,284.818,-107.496,172.142,39.272,157.467
C08327=1047.383,285.065,-107.527,172.145,39.275,157.467
C08328=1047.389,285.313,-107.558,172.148,39.278,157.468
C08329=1047.396,285.561,-107.590,172.152,39.281,157.469
C08330=1047.403,285.808,-107.621,172.154,39.284,157.470
C08331=1047.410,286.056,-107.653,172.158,39.287,157.470
C08332=1047.416,286.305,-107.685,172.161,39.289,157.471
C08333=1047.422,286.552,-107.716,172.164,39.292,157.472
C08334=1047.429,286.800,-107.748,172.167,39.295,157.472
C08335=1047.436,287.048,-107.779,172.171,39.298,157.473
C08336=1047.443,287.296,-107.810,172.174,39.301,157.474
C08337=1047.449,287.544,-107.842,172.177,39.304,157.475
C08338=1047.456,287.792,-107.873,172.181,39.307,157.475
C08339=1047.463,288.040,-107.905,172.184,39.310,157.476
C08340=1047.469,288.288,-107.937,172.187,39.313,157.477
C08341=1047.475,288.536,-107.968,172.190,39.316,157.478
C08342=1047.482,288.783,-108.000,172.194,39.318,157.478
C08343=1047.489,289.031,-108.032,172.196,39.321,157.479
C08344=1047.495,289.279,-108.064,172.200,39.325,157.480
C08345=1047.502,289.527,-108.095,172.203,39.327,157.481
C08346=1047.509,289.775,-108.127,172.207,39.330,157.481
C08347=1047.516,290.023,-108.159,172.210,39.334,157.482
C08348=1047.522,290.271,-108.191,172.213,39.336,157.483
C08349=1047.530,290.556,-108.228,172.217,39.340,157.484
C08350=1047.537,290.840,-108.264,172.221,39.343,157.485
C08351=1047.545,291.125,-108.301,172.225,39.346,157.486
C08352=1047.553,291.410,-108.338,172.228,39.350,157.486
C08353=1047.559,291.657,-108.369,172.232,39.353,157.487
C08354=1047.566,291.906,-108.402,172.235,39.356,157.488
C08355=1047.573,292.154,-108.434,172.239,39.359,157.489
C08356=1047.579,292.402,-108.466,172.241,39.362,157.490
C08357=1047.586,292.649,-108.498,172.245,39.365,157.490
C08358=1047.593,292.897,-108.529,172.249,39.367,157.491
C08359=1047.599,293.145,-108.562,172.252,39.371,157.492
C08360=1047.606,293.393,-108.593,172.255,39.374,157.493
C08361=1047.612,293.640,-108.625,172.258,39.376,157.493
C08362=1047.619,293.889,-108.658,172.262,39.380,157.494
C08363=1047.626,294.136,-108.690,172.266,39.383,157.495
C08364=1047.632,294.384,-108.722,172.268,39.385,157.496
C08365=1047.639,294.631,-108.754,172.272,39.389,157.496
C08366=1047.645,294.880,-108.786,172.276,39.391,157.497
C08367=1047.652,295.127,-108.819,172.279,39.395,157.498
C08368=1047.659,295.376,-108.851,172.282,39.398,157.499
C08369=1047.666,295.623,-108.883,172.286,39.400,157.499
C08370=1047.672,295.871,-108.916,172.289,39.404,157.500
C08371=1047.679,296.119,-108.947,172.292,39.406,157.501
C08372=1047.685,296.366,-108.980,172.296,39.410,157.502
C08373=1047.692,296.614,-109.013,172.299,39.413,157.503
C08374=1047.699,296.861,-109.045,172.303,39.416,157.503
C08375=1047.706,297.109,-109.078,172.306,39.419,157.504
C08376=1047.712,297.358,-109.110,172.309,39.422,157.505
C08377=1047.718,297.605,-109.143,172.313,39.425,157.506
C08378=1047.724,297.853,-109.175,172.316,39.428,157.507
C08379=1047.731,298.100,-109.208,172.320,39.431,157.508
C08380=1047.737,298.348,-109.240,172.324,39.435,157.508
C08381=1047.744,298.596,-109.273,172.326,39.438,157.509
C08382=1047.751,298.844,-109.306,172.330,39.441,157.510
C08383=1047.757,299.092,-109.338,172.334,39.444,157.511
C08384=1047.764,299.339,-109.370,172.337,39.447,157.512
C08385=1047.771,299.587,-109.404,172.340,39.450,157.512
C08386=1047.777,299.835,-109.436,172.344,39.453,157.513
C08387=1047.783,300.083,-109.469,172.348,39.456,157.514
C08388=1047.789,300.330,-109.502,172.351,39.460,157.515
C08389=1047.797,300.578,-109.534,172.355,39.462,157.516
C08390=1047.803,300.826,-109.567,172.358,39.466,157.516
C08391=1047.810,301.073,-109.600,172.361,39.469,157.517
C08392=1047.816,301.321,-109.632,172.365,39.472,157.518
C08393=1047.823,301.569,-109.666,172.369,39.475,157.519
C08394=1047.829,301.817,-109.698,172.372,39.478,157.520
C08395=1047.836,302.063,-109.731,172.375,39.481,157.520
C08396=1047.843,302.312,-109.764,172.379,39.485,157.521
C08397=1047.850,302.559,-109.797,172.383,39.487,157.522
C08398=1047.856,302.807,-109.830,172.387,39.491,157.523
C08399=1047.863,303.055,-109.863,172.390,39.494,157.524
C08400=1047.869,303.303,-109.896,172.393,39.497,157.525
C08401=1047.876,303.550,-109.928,172.397,39.500,157.525
C08402=1047.883,303.798,-109.962,172.401,39.503,157.526
C08403=1047.890,304.045,-109.994,172.404,39.507,157.527
C08404=1047.897,304.294,-110.027,172.407,39.510,157.528
C08405=1047.904,304.594,-110.067,172.411,39.513,157.529
C08406=1047.912,304.895,-110.108,172.416,39.517,157.530
C08407=1047.921,305.196,-110.147,172.420,39.521,157.531
C08408=1047.929,305.498,-110.187,172.425,39.525,157.532
C08409=1047.936,305.744,-110.221,172.428,39.528,157.533
C08410=1047.943,305.993,-110.254,172.432,39.532,157.534
C08411=1047.949,306.240,-110.287,172.436,39.534,157.534
C08412=1047.956,306.488,-110.320,172.440,39.538,157.535
C08413=1047.963,306.736,-110.353,172.443,39.541,157.536
C08414=1047.970,306.983,-110.387,172.447,39.544,157.537
C08415=1047.977,307.231,-110.419,172.450,39.547,157.538
C08416=1047.984,307.479,-110.452,172.454,39.550,157.539
C08417=1047.990,307.726,-110.486,172.458,39.554,157.539
C08418=1047.997,307.974,-110.519,172.462,39.557,157.540
C08419=1048.004,308.221,-110.552,172.465,39.560,157.541
C08420=1048.011,308.469,-110.585,172.469,39.563,157.542
C08421=1048.017,308.716,-110.619,172.473,39.566,157.543
C08422=1048.024,308.965,-110.652,172.476,39.570,157.544
C08423=1048.031,309.212,-110.686,172.480,39.573,157.544
C08424=1048.038,309.460,-110.718,172.483,39.576,157.545
C08425=1048.046,309.707,-110.752,172.487,39.579,157.546
C08426=1048.052,309.955,-110.784,172.491,39.582,157.547
C08427=1048.059,310.203,-110.818,172.495,39.585,157.548
C08428=1048.066,310.450,-110.852,172.499,39.589,157.549
C08429=1048.073,310.698,-110.885,172.503,39.592,157.550
C08430=1048.080,310.946,-110.919,172.506,39.595,157.550
C08431=1048.086,311.193,-110.951,172.509,39.598,157.551
C08432=1048.093,311.441,-110.985,172.513,39.601,157.552
C08433=1048.100,311.688,-111.019,172.517,39.605,157.553
C08434=1048.107,311.935,-111.053,172.521,39.608,157.554
C08435=1048.114,312.184,-111.086,172.525,39.611,157.555
C08436=1048.121,312.431,-111.119,172.529,39.615,157.556
C08437=1048.128,312.679,-111.153,172.532,39.618,157.556
C08438=1048.135,312.927,-111.186,172.536,39.621,157.557
C08439=1048.142,313.174,-111.220,172.540,39.624,157.558
C08440=1048.148,313.422,-111.254,172.544,39.628,157.559
C08441=1048.155,313.669,-111.288,172.548,39.631,157.560
C08442=1048.161,313.917,-111.322,172.552,39.634,157.561
C08443=1048.168,314.164,-111.356,172.555,39.638,157.562
C08444=1048.174,314.412,-111.390,172.559,39.641,157.563
C08445=1048.182,314.660,-111.424,172.562,39.645,157.564
C08446=1048.188,314.907,-111.457,172.566,39.648,157.564
C08447=1048.195,315.155,-111.492,172.570,39.651,157.565
C08448=1048.202,315.403,-111.526,172.574,39.655,157.566
C08449=1048.208,315.650,-111.560,172.578,39.658,157.567
C08450=1048.215,315.898,-111.593,172.582,39.662,157.568
C08451=1048.221,316.145,-111.628,172.586,39.665,157.569
C08452=1048.228,316.392,-111.662,172.590,39.668,157.570
C08453=1048.235,316.640,-111.696,172.594,39.672,157.571
C08454=1048.242,316.887,-111.730,172.598,39.675,157.572
C08455=1048.248,317.135,-111.765,172.601,39.679,157.573
C08456=1048.255,317.382,-111.798,172.605,39.682,157.574
C08457=1048.261,317.630,-111.833,172.609,39.685,157.574
C08458=1048.268,317.878,-111.868,172.613,39.689,157.575
C08459=1048.275,318.125,-111.902,172.616,39.692,157.576
C08460=1048.281,318.373,-111.936,172.620,39.696,157.577
C08461=1048.290,318.678,-111.978,172.625,39.700,157.578
C08462=1048.299,318.984,-112.020,172.630,39.704,157.579
C08463=1048.307,319.289,-112.062,172.635,39.709,157.581
C08464=1048.316,319.594,-112.105,172.640,39.713,157.582
C08465=1048.322,319.842,-112.139,172.643,39.716,157.583
C08466=1048.329,320.090,-112.173,172.647,39.720,157.584
C08467=1048.336,320.337,-112.208,172.651,39.724,157.585
C08468=1048.343,320.585,-112.242,172.655,39.727,157.585
C08469=1048.350,320.833,-112.276,172.659,39.730,157.586
C08470=1048.356,321.080,-112.311,172.663,39.734,157.587
C08471=1048.363,321.327,-112.345,172.667,39.737,157.588
C08472=1048.370,321.575,-112.380,172.672,39.740,157.589
C08473=1048.377,321.822,-112.414,172.676,39.744,157.590
C08474=1048.384,322.070,-112.449,172.680,39.747,157.591
C08475=1048.391,322.317,-112.483,172.684,39.751,157.592
C08476=1048.398,322.565,-112.518,172.688,39.755,157.593
C08477=1048.404,322.813,-112.552,172.692,39.758,157.594
C08478=1048.412,323.060,-112.587,172.696,39.762,157.595
C08479=1048.418,323.308,-112.621,172.699,39.765,157.596
C08480=1048.426,323.555,-112.656,172.704,39.769,157.597
C08481=1048.432,323.803,-112.690,172.707,39.772,157.598
C08482=1048.439,324.050,-112.725,172.711,39.776,157.599
C08483=1048.446,324.297,-112.760,172.715,39.779,157.600
C08484=1048.453,324.545,-112.794,172.719,39.783,157.601
C08485=1048.460,324.792,-112.829,172.724,39.786,157.602
C08486=1048.467,325.040,-112.864,172.728,39.790,157.603
C08487=1048.474,325.288,-112.899,172.732,39.793,157.603
C08488=1048.482,325.535,-112.933,172.736,39.797,157.604
C08489=1048.488,325.783,-112.969,172.740,39.800,157.605
C08490=1048.496,326.030,-113.003,172.744,39.804,157.606
C08491=1048.502,326.278,-113.038,172.748,39.807,157.607
C08492=1048.509,326.525,-113.073,172.753,39.811,157.608
C08493=1048.517,326.772,-113.107,172.757,39.814,157.609
C08494=1048.523,327.020,-113.142,172.761,39.818,157.610
C08495=1048.531,327.267,-113.176,172.765,39.822,157.611
C08496=1048.538,327.515,-113.212,172.769,39.825,157.612
C08497=1048.545,327.763,-113.247,172.773,39.829,157.613
C08498=1048.552,328.010,-113.281,172.778,39.832,157.614
C08499=1048.559,328.257,-113.316,172.782,39.836,157.615
C08500=1048.566,328.505,-113.352,172.786,39.840,157.616
C08501=1048.574,328.752,-113.387,172.790,39.843,157.617
C08502=1048.581,329.000,-113.422,172.794,39.847,157.618
C08503=1048.588,329.247,-113.457,172.799,39.851,157.619
C08504=1048.595,329.494,-113.491,172.803,39.854,157.620
C08505=1048.602,329.742,-113.527,172.807,39.858,157.621
C08506=1048.609,329.989,-113.562,172.811,39.862,157.622
C08507=1048.616,330.237,-113.597,172.815,39.865,157.623
C08508=1048.623,330.484,-113.632,172.820,39.869,157.624
C08509=1048.629,330.732,-113.667,172.824,39.873,157.625
C08510=1048.637,330.979,-113.704,172.828,39.876,157.626
C08511=1048.644,331.226,-113.739,172.832,39.880,157.627
C08512=1048.651,331.474,-113.774,172.836,39.884,157.628
C08513=1048.657,331.721,-113.809,172.841,39.888,157.629
C08514=1048.665,331.969,-113.844,172.845,39.891,157.630
C08515=1048.672,332.216,-113.880,172.849,39.895,157.631
C08516=1048.679,332.463,-113.915,172.853,39.899,157.632
C08517=1048.687,332.764,-113.959,172.858,39.903,157.633
C08518=1048.696,333.065,-114.002,172.864,39.908,157.635
C08519=1048.704,333.364,-114.045,172.869,39.912,157.636
C08520=1048.713,333.665,-114.088,172.874,39.917,157.637
C08521=1048.719,333.912,-114.123,172.878,39.921,157.638
C08522=1048.727,334.160,-114.160,172.883,39.925,157.639
C08523=1048.733,334.407,-114.195,172.887,39.929,157.640
C08524=1048.740,334.654,-114.231,172.891,39.933,157.641
C08525=1048.748,334.902,-114.267,172.896,39.936,157.642
C08526=1048.755,335.149,-114.302,172.901,39.940,157.644
C08527=1048.762,335.397,-114.338,172.905,39.944,157.645
C08528=1048.769,335.644,-114.374,172.909,39.948,157.646
C08529=1048.776,335.892,-114.409,172.914,39.951,157.647
C08530=1048.784,336.139,-114.445,172.918,39.956,157.648
C08531=1048.790,336.386,-114.481,172.922,39.960,157.649
C08532=1048.797,336.634,-114.517,172.927,39.963,157.650
C08533=1048.804,336.880,-114.553,172.931,39.967,157.651
C08534=1048.812,337.129,-114.588,172.935,39.971,157.652
C08535=1048.818,337.376,-114.625,172.940,39.975,157.653
C08536=1048.825,337.622,-114.661,172.945,39.979,157.654
C08537=1048.833,337.870,-114.697,172.949,39.983,157.655
C08538=1048.839,338.117,-114.733,172.954,39.987,157.656
C08539=1048.846,338.365,-114.769,172.958,39.991,157.657
C08540=1048.854,338.612,-114.805,172.962,39.995,157.659
C08541=1048.861,338.859,-114.842,172.967,39.999,157.660
C08542=1048.868,339.106,-114.877,172.971,40.003,157.661
C08543=1048.875,339.354,-114.913,172.975,40.006,157.662
C08544=1048.881,339.601,-114.949,172.980,40.011,157.663
C08545=1048.889,339.849,-114.986,172.985,40.015,157.664
C08546=1048.896,340.095,-115.021,172.989,40.018,157.665
C08547=1048.903,340.343,-115.058,172.994,40.023,157.666
C08548=1048.910,340.590,-115.094,172.998,40.026,157.667
C08549=1048.918,340.837,-115.130,173.003,40.031,157.669
C08550=1048.925,341.085,-115.167,173.007,40.034,157.670
C08551=1048.932,341.332,-115.203,173.011,40.039,157.671
C08552=1048.939,341.579,-115.239,173.017,40.042,157.672
C08553=1048.946,341.826,-115.276,173.021,40.047,157.673
C08554=1048.953,342.074,-115.312,173.026,40.051,157.674
C08555=1048.960,342.322,-115.349,173.030,40.055,157.675
C08556=1048.967,342.568,-115.385,173.035,40.059,157.676
C08557=1048.974,342.816,-115.421,173.039,40.063,157.677
C08558=1048.982,343.063,-115.458,173.043,40.067,157.679
C08559=1048.989,343.310,-115.495,173.049,40.071,157.680
C08560=1048.996,343.557,-115.531,173.053,40.075,157.681
C08561=1049.003,343.805,-115.568,173.058,40.079,157.682
C08562=1049.011,344.051,-115.604,173.062,40.083,157.683
C08563=1049.018,344.299,-115.641,173.067,40.088,157.684
C08564=1049.025,344.547,-115.678,173.072,40.091,157.685
C08565=1049.032,344.793,-115.714,173.077,40.096,157.687
C08566=1049.039,345.041,-115.751,173.081,40.100,157.688
C08567=1049.047,345.288,-115.788,173.086,40.104,157.689
C08568=1049.053,345.535,-115.825,173.090,40.108,157.690
C08569=1049.060,345.782,-115.862,173.096,40.112,157.691
C08570=1049.068,346.029,-115.898,173.100,40.117,157.692
C08571=1049.075,346.277,-115.935,173.105,40.121,157.694
C08572=1049.082,346.523,-115.972,173.109,40.125,157.695
C08573=1049.091,346.820,-116.016,173.115,40.130,157.696
C08574=1049.099,347.117,-116.061,173.121,40.135,157.698
C08575=1049.108,347.414,-116.104,173.127,40.140,157.699
C08576=1049.117,347.709,-116.149,173.132,40.146,157.701
C08577=1049.123,347.957,-116.186,173.137,40.149,157.702
C08578=1049.131,348.204,-116.223,173.142,40.154,157.703
C08579=1049.139,348.451,-116.261,173.147,40.158,157.704
C08580=1049.146,348.699,-116.297,173.151,40.162,157.705
C08581=1049.153,348.946,-116.335,173.156,40.166,157.706
C08582=1049.160,349.192,-116.372,173.161,40.171,157.708
C08583=1049.167,349.440,-116.408,173.166,40.175,157.709
C08584=1049.174,349.687,-116.446,173.171,40.179,157.710
C08585=1049.182,349.934,-116.483,173.175,40.183,157.711
C08586=1049.190,350.181,-116.520,173.181,40.188,157.712
C08587=1049.197,350.428,-116.558,173.185,40.193,157.714
C08588=1049.204,350.676,-116.595,173.190,40.197,157.715
C08589=1049.211,350.923,-116.632,173.195,40.201,157.716
C08590=1049.218,351.170,-116.670,173.200,40.205,157.717
C08591=1049.226,351.417,-116.707,173.205,40.210,157.719
C08592=1049.234,351.664,-116.744,173.209,40.214,157.720
C08593=1049.241,351.911,-116.782,173.215,40.219,157.721
C08594=1049.248,352.158,-116.819,173.220,40.223,157.722
C08595=1049.255,352.405,-116.856,173.224,40.227,157.724
C08596=1049.262,352.652,-116.894,173.230,40.232,157.725
C08597=1049.269,352.899,-116.931,173.234,40.236,157.726
C08598=1049.276,353.146,-116.969,173.239,40.241,157.727
C08599=1049.284,353.393,-117.007,173.245,40.245,157.729
C08600=1049.291,353.640,-117.045,173.249,40.250,157.730
C08601=1049.299,353.888,-117.083,173.254,40.254,157.731
C08602=1049.306,354.135,-117.120,173.260,40.259,157.733
C08603=1049.314,354.382,-117.158,173.264,40.263,157.734
C08604=1049.321,354.629,-117.196,173.269,40.268,157.735
C08605=1049.328,354.876,-117.233,173.274,40.272,157.736
C08606=1049.336,355.123,-117.271,173.280,40.277,157.738
C08607=1049.343,355.370,-117.308,173.284,40.281,157.739
C08608=1049.350,355.617,-117.347,173.290,40.286,157.740
C08609=1049.358,355.864,-117.384,173.295,40.290,157.741
C08610=1049.365,356.111,-117.422,173.299,40.295,157.743
C08611=1049.372,356.357,-117.460,173.305,40.299,157.744
C08612=1049.380,356.605,-117.498,173.310,40.304,157.745
C08613=1049.388,356.852,-117.536,173.315,40.308,157.747
C08614=1049.395,357.099,-117.574,173.320,40.313,157.748
C08615=1049.402,357.346,-117.611,173.325,40.317,157.749
C08616=1049.410,357.592,-117.649,173.330,40.322,157.751
C08617=1049.417,357.840,-117.689,173.336,40.327,157.752
C08618=1049.425,358.087,-117.726,173.340,40.332,157.753
C08619=1049.432,358.334,-117.764,173.346,40.336,157.754
C08620=1049.439,358.581,-117.802,173.351,40.341,157.756
C08621=1049.447,358.827,-117.840,173.357,40.345,157.757
C08622=1049.454,359.075,-117.879,173.362,40.350,157.759
C08623=1049.462,359.322,-117.917,173.366,40.355,157.760
C08624=1049.469,359.568,-117.955,173.372,40.359,157.761
C08625=1049.477,359.815,-117.993,173.377,40.364,157.763
C08626=1049.485,360.062,-118.032,173.383,40.369,157.764
C08627=1049.491,360.310,-118.070,173.388,40.374,157.765
C08628=1049.499,360.556,-118.108,173.392,40.378,157.767
C08629=1049.509,360.858,-118.155,173.399,40.384,157.768
C08630=1049.517,361.160,-118.202,173.406,40.390,157.770
C08631=1049.527,361.462,-118.249,173.412,40.396,157.772
C08632=1049.536,361.764,-118.297,173.419,40.402,157.773
C08633=1049.543,362.011,-118.335,173.424,40.406,157.775
C08634=1049.551,362.257,-118.373,173.430,40.411,157.776
C08635=1049.558,362.505,-118.412,173.435,40.416,157.777
C08636=1049.566,362.751,-118.451,173.440,40.421,157.779
C08637=1049.574,362.998,-118.489,173.446,40.425,157.780
C08638=1049.581,363.245,-118.528,173.450,40.430,157.782
C08639=1049.588,363.492,-118.566,173.456,40.436,157.783
C08640=1049.596,363.739,-118.605,173.461,40.440,157.784
C08641=1049.604,363.985,-118.644,173.467,40.445,157.786
C08642=1049.611,364.233,-118.684,173.473,40.450,157.787
C08643=1049.619,364.479,-118.722,173.478,40.455,157.789
C08644=1049.626,364.727,-118.761,173.483,40.460,157.790
C08645=1049.634,364.973,-118.800,173.489,40.465,157.792
C08646=1049.641,365.219,-118.839,173.495,40.470,157.793
C08647=1049.648,365.467,-118.878,173.500,40.475,157.794
C08648=1049.656,365.713,-118.917,173.506,40.480,157.796
C08649=1049.663,365.960,-118.956,173.510,40.485,157.797
C08650=1049.671,366.207,-118.994,173.516,40.490,157.799
C08651=1049.679,366.454,-119.034,173.521,40.495,157.800
C08652=1049.686,366.700,-119.073,173.527,40.500,157.802
C08653=1049.694,366.947,-119.112,173.532,40.505,157.803
C08654=1049.702,367.194,-119.151,173.538,40.510,157.805
C08655=1049.709,367.441,-119.191,173.544,40.515,157.806
C08656=1049.717,367.688,-119.230,173.549,40.520,157.808
C08657=1049.725,367.934,-119.269,173.555,40.525,157.809
C08658=1049.732,368.182,-119.308,173.560,40.530,157.810
C08659=1049.740,368.428,-119.347,173.566,40.535,157.812
C08660=1049.748,368.674,-119.387,173.572,40.541,157.814
C08661=1049.756,368.922,-119.426,173.577,40.545,157.815
C08662=1049.763,369.169,-119.465,173.583,40.551,157.816
C08663=1049.770,369.415,-119.505,173.589,40.556,157.818
C08664=1049.779,369.662,-119.544,173.595,40.561,157.819
C08665=1049.786,369.909,-119.584,173.601,40.566,157.821
C08666=1049.794,370.155,-119.622,173.606,40.571,157.822
C08667=1049.802,370.402,-119.662,173.612,40.576,157.824
C08668=1049.810,370.649,-119.702,173.617,40.582,157.825
C08669=1049.818,370.896,-119.741,173.623,40.587,157.827
C08670=1049.825,371.142,-119.780,173.629,40.592,157.828
C08671=1049.833,371.389,-119.820,173.634,40.597,157.830
C08672=1049.841,371.635,-119.860,173.640,40.602,157.831
C08673=1049.849,371.882,-119.900,173.646,40.607,157.833
C08674=1049.856,372.129,-119.939,173.652,40.613,157.835
C08675=1049.864,372.375,-119.979,173.658,40.618,157.836
C08676=1049.871,372.622,-120.019,173.664,40.624,157.838
C08677=1049.879,372.869,-120.060,173.669,40.629,157.839
C08678=1049.887,373.116,-120.100,173.675,40.634,157.841
C08679=1049.894,373.362,-120.139,173.681,40.639,157.842
C08680=1049.902,373.609,-120.179,173.687,40.645,157.844
C08681=1049.910,373.856,-120.219,173.692,40.651,157.846
C08682=1049.918,374.102,-120.260,173.699,40.656,157.847
C08683=1049.926,374.348,-120.299,173.705,40.661,157.849
C08684=1049.934,374.595,-120.339,173.711,40.667,157.850
C08685=1049.944,374.936,-120.394,173.719,40.674,157.853
C08686=1049.954,375.277,-120.450,173.727,40.681,157.855
C08687=1049.966,375.617,-120.505,173.735,40.689,157.857
C08688=1049.977,375.958,-120.561,173.743,40.697,157.859
C08689=1049.984,376.205,-120.601,173.749,40.702,157.861
C08690=1049.992,376.451,-120.642,173.756,40.708,157.863
C08691=1050.000,376.698,-120.682,173.762,40.713,157.864
C08692=1050.009,376.944,-120.722,173.767,40.719,157.866
C08693=1050.017,377.191,-120.762,173.773,40.724,157.867
C08694=1050.024,377.437,-120.802,173.780,40.730,157.869
C08695=1050.033,377.684,-120.843,173.786,40.735,157.871
C08696=1050.040,377.931,-120.883,173.792,40.741,157.872
C08697=1050.048,378.167,-120.922,173.797,40.746,157.874
C08698=1050.055,378.403,-120.961,173.804,40.751,157.876
C08699=1050.063,378.641,-121.000,173.810,40.757,157.877
C08700=1050.071,378.877,-121.039,173.815,40.762,157.879
C08701=1050.078,379.113,-121.077,173.821,40.768,157.880
C08702=1050.086,379.351,-121.116,173.827,40.774,157.882
C08703=1050.094,379.587,-121.155,173.833,40.779,157.884
C08704=1050.102,379.824,-121.195,173.839,40.784,157.885
C08705=1050.110,380.070,-121.235,173.845,40.790,157.887
C08706=1050.118,380.317,-121.276,173.851,40.795,157.889
C08707=1050.125,380.563,-121.317,173.858,40.801,157.890
C08708=1050.133,380.810,-121.358,173.864,40.807,157.892
C08709=1050.141,381.056,-121.399,173.870,40.813,157.894
C08710=1050.148,381.302,-121.440,173.877,40.819,157.896
C08711=1050.157,381.549,-121.481,173.883,40.825,157.897
C08712=1050.165,381.796,-121.521,173.889,40.830,157.899
C08713=1050.173,382.042,-121.562,173.896,40.836,157.901
C08714=1050.181,382.288,-121.604,173.902,40.842,157.903
C08715=1050.189,382.535,-121.645,173.909,40.848,157.904
C08716=1050.197,382.781,-121.686,173.914,40.854,157.906
C08717=1050.205,383.028,-121.727,173.920,40.860,157.908
C08718=1050.213,383.273,-121.768,173.927,40.866,157.910
C08719=1050.222,383.520,-121.809,173.933,40.871,157.911
C08720=1050.229,383.767,-121.850,173.940,40.878,157.913
C08721=1050.237,384.013,-121.892,173.946,40.883,157.915
C08722=1050.246,384.260,-121.933,173.953,40.889,157.917
C08723=1050.253,384.506,-121.974,173.959,40.895,157.919
C08724=1050.261,384.752,-122.015,173.966,40.901,157.920
C08725=1050.270,384.999,-122.056,173.972,40.907,157.922
C08726=1050.278,385.245,-122.098,173.979,40.914,157.924
C08727=1050.287,385.491,-122.140,173.985,40.919,157.926
C08728=1050.294,385.738,-122.181,173.992,40.925,157.928
C08729=1050.303,385.984,-122.223,173.998,40.931,157.929
C08730=1050.311,386.231,-122.264,174.005,40.937,157.931
C08731=1050.319,386.477,-122.306,174.011,40.944,157.933
C08732=1050.327,386.723,-122.347,174.019,40.950,157.935
C08733=1050.336,386.970,-122.388,174.026,40.955,157.937
C08734=1050.344,387.216,-122.430,174.032,40.962,157.939
C08735=1050.353,387.462,-122.472,174.039,40.968,157.940
C08736=1050.360,387.708,-122.514,174.045,40.974,157.942
C08737=1050.369,387.955,-122.556,174.052,40.980,157.944
C08738=1050.377,388.201,-122.596,174.059,40.987,157.946
C08739=1050.385,388.448,-122.639,174.065,40.993,157.948
C08740=1050.394,388.694,-122.680,174.072,40.999,157.950
C08741=1050.406,389.048,-122.741,174.082,41.008,157.953
C08742=1050.418,389.400,-122.800,174.091,41.017,157.955
C08743=1050.430,389.754,-122.861,174.101,41.026,157.958
C08744=1050.441,390.108,-122.922,174.111,41.035,157.961
C08745=1050.450,390.354,-122.964,174.118,41.041,157.963
C08746=1050.459,390.601,-123.006,174.125,41.048,157.965
C08747=1050.466,390.847,-123.047,174.132,41.054,157.967
C08748=1050.475,391.092,-123.090,174.138,41.061,157.969
C08749=1050.484,391.339,-123.132,174.145,41.067,157.970
C08750=1050.492,391.586,-123.175,174.153,41.073,157.973
C08751=1050.500,391.831,-123.217,174.160,41.080,157.974
C08752=1050.509,392.077,-123.259,174.166,41.086,157.976
C08753=1050.517,392.324,-123.301,174.173,41.092,157.978
C08754=1050.525,392.570,-123.344,174.181,41.099,157.980
C08755=1050.534,392.816,-123.386,174.188,41.105,157.982
C08756=1050.542,393.062,-123.429,174.194,41.112,157.984
C08757=1050.550,393.309,-123.471,174.201,41.119,157.986
C08758=1050.559,393.555,-123.514,174.209,41.125,157.988
C08759=1050.567,393.801,-123.557,174.216,41.132,157.990
C08760=1050.576,394.047,-123.599,174.223,41.138,157.992
C08761=1050.584,394.292,-123.641,174.229,41.145,157.994
C08762=1050.593,394.538,-123.684,174.237,41.152,157.997
C08763=1050.601,394.785,-123.727,174.244,41.158,157.999
C08764=1050.609,395.031,-123.770,174.251,41.165,158.001
C08765=1050.618,395.277,-123.813,174.259,41.172,158.003
C08766=1050.626,395.523,-123.856,174.266,41.178,158.005
C08767=1050.636,395.769,-123.898,174.273,41.185,158.007
C08768=1050.644,396.015,-123.941,174.281,41.192,158.009
C08769=1050.652,396.262,-123.984,174.287,41.198,158.011
C08770=1050.661,396.508,-124.027,174.295,41.205,158.013
C08771=1050.669,396.754,-124.070,174.302,41.212,158.015
C08772=1050.678,397.000,-124.113,174.309,41.219,158.017
C08773=1050.687,397.245,-124.156,174.317,41.226,158.019
C08774=1050.695,397.491,-124.199,174.324,41.233,158.022
C08775=1050.704,397.737,-124.242,174.332,41.239,158.024
C08776=1050.713,397.984,-124.286,174.339,41.246,158.026
C08777=1050.721,398.230,-124.329,174.347,41.253,158.028
C08778=1050.730,398.476,-124.372,174.354,41.260,158.030
C08779=1050.739,398.722,-124.416,174.361,41.267,158.032
C08780=1050.746,398.968,-124.459,174.369,41.274,158.035
C08781=1050.755,399.214,-124.502,174.376,41.281,158.037
C08782=1050.764,399.460,-124.546,174.384,41.288,158.039
C08783=1050.773,399.706,-124.589,174.391,41.295,158.041
C08784=1050.782,399.952,-124.633,174.399,41.302,158.043
C08785=1050.790,400.198,-124.676,174.406,41.309,158.045
C08786=1050.799,400.445,-124.720,174.414,41.316,158.048
C08787=1050.808,400.690,-124.763,174.422,41.323,158.050
C08788=1050.817,400.935,-124.807,174.429,41.331,158.052
C08789=1050.826,401.182,-124.850,174.438,41.338,158.054
C08790=1050.834,401.428,-124.895,174.445,41.345,158.057
C08791=1050.842,401.674,-124.938,174.453,41.352,158.059
C08792=1050.852,401.920,-124.982,174.460,41.359,158.061
C08793=1050.861,402.166,-125.026,174.468,41.366,158.063
C08794=1050.870,402.412,-125.070,174.476,41.373,158.066
C08795=1050.878,402.658,-125.113,174.483,41.380,158.068
C08796=1050.887,402.904,-125.157,174.491,41.388,158.070
C08797=1050.901,403.276,-125.224,174.503,41.399,158.074
C08798=1050.913,403.648,-125.291,174.515,41.410,158.077
C08799=1050.927,404.020,-125.357,174.527,41.421,158.081
C08800=1050.940,404.391,-125.424,174.539,41.432,158.084
C08801=1050.950,404.637,-125.468,174.547,41.439,158.086
C08802=1050.958,404.884,-125.513,174.554,41.447,158.089
C08803=1050.967,405.129,-125.557,174.563,41.455,158.091
C08804=1050.976,405.375,-125.602,174.571,41.462,158.094
C08805=1050.984,405.621,-125.647,174.579,41.469,158.096
C08806=1050.994,405.867,-125.691,174.588,41.477,158.098
C08807=1051.002,406.113,-125.735,174.595,41.485,158.101
C08808=1051.011,406.358,-125.780,174.603,41.492,158.103
C08809=1051.020,406.605,-125.825,174.612,41.500,158.106
C08810=1051.030,406.850,-125.869,174.620,41.507,158.108
C08811=1051.038,407.096,-125.914,174.628,41.515,158.110
C08812=1051.048,407.342,-125.958,174.636,41.523,158.113
C08813=1051.056,407.588,-126.003,174.644,41.530,158.115
C08814=1051.066,407.833,-126.048,174.652,41.538,158.118
C08815=1051.074,408.079,-126.092,174.661,41.546,158.120
C08816=1051.083,408.325,-126.138,174.669,41.554,158.123
C08817=1051.093,408.571,-126.183,174.678,41.561,158.125
C08818=1051.101,408.817,-126.227,174.686,41.569,158.128
C08819=1051.111,409.063,-126.272,174.695,41.577,158.130
C08820=1051.120,409.308,-126.318,174.703,41.585,158.133
C08821=1051.129,409.554,-126.363,174.711,41.592,158.135
C08822=1051.138,409.800,-126.407,174.720,41.601,158.138
C08823=1051.147,410.046,-126.452,174.728,41.608,158.140
C08824=1051.157,410.292,-126.497,174.736,41.616,158.143
C08825=1051.166,410.537,-126.543,174.745,41.624,158.145
C08826=1051.175,410.783,-126.588,174.753,41.632,158.148
C08827=1051.185,411.029,-126.633,174.762,41.640,158.150
C08828=1051.194,411.275,-126.678,174.771,41.648,158.153
C08829=1051.204,411.520,-126.723,174.779,41.656,158.156
C08830=1051.213,411.766,-126.769,174.789,41.664,158.158
C08831=1051.222,412.011,-126.815,174.797,41.672,158.161
C08832=1051.232,412.257,-126.860,174.806,41.680,158.163
C08833=1051.240,412.503,-126.905,174.815,41.688,158.166
C08834=1051.250,412.749,-126.951,174.823,41.696,158.169
C08835=1051.260,412.995,-126.996,174.832,41.704,158.171
C08836=1051.269,413.240,-127.042,174.841,41.712,158.174
C08837=1051.278,413.486,-127.087,174.850,41.721,158.177
C08838=1051.287,413.731,-127.133,174.858,41.729,158.179
C08839=1051.297,413.977,-127.179,174.867,41.737,158.182
C08840=1051.306,414.223,-127.225,174.877,41.745,158.185
C08841=1051.315,414.468,-127.271,174.885,41.754,158.187
C08842=1051.324,414.714,-127.317,174.894,41.762,158.190
C08843=1051.334,414.959,-127.363,174.903,41.770,158.193
C08844=1051.343,415.205,-127.409,174.913,41.779,158.196
C08845=1051.353,415.450,-127.455,174.922,41.787,158.198
C08846=1051.362,415.696,-127.501,174.931,41.795,158.201
C08847=1051.372,415.942,-127.547,174.939,41.804,158.204
C08848=1051.381,416.187,-127.594,174.949,41.813,158.207
C08849=1051.392,416.432,-127.640,174.958,41.821,158.209
C08850=1051.401,416.678,-127.686,174.967,41.829,158.212
C08851=1051.411,416.923,-127.732,174.977,41.838,158.215
C08852=1051.420,417.169,-127.778,174.986,41.846,158.218
C08853=1051.435,417.548,-127.850,175.000,41.860,158.222
C08854=1051.449,417.926,-127.921,175.014,41.873,158.226
C08855=1051.464,418.305,-127.993,175.030,41.886,158.231
C08856=1051.480,418.684,-128.065,175.044,41.900,158.235
C08857=1051.489,418.929,-128.111,175.053,41.908,158.238
C08858=1051.499,419.175,-128.158,175.063,41.917,158.241
C08859=1051.509,419.420,-128.205,175.073,41.926,158.244
C08860=1051.518,419.665,-128.251,175.082,41.935,158.247
C08861=1051.528,419.911,-128.299,175.091,41.944,158.250
C08862=1051.538,420.157,-128.345,175.101,41.952,158.253
C08863=1051.547,420.401,-128.392,175.112,41.961,158.256
C08864=1051.557,420.646,-128.440,175.121,41.970,158.259
C08865=1051.566,420.893,-128.487,175.131,41.979,158.262
C08866=1051.577,421.138,-128.534,175.140,41.988,158.265
C08867=1051.586,421.383,-128.581,175.150,41.997,158.268
C08868=1051.596,421.628,-128.629,175.161,42.006,158.271
C08869=1051.606,421.873,-128.676,175.170,42.015,158.274
C08870=1051.616,422.119,-128.722,175.180,42.024,158.277
C08871=1051.626,422.365,-128.769,175.190,42.034,158.280
C08872=1051.635,422.610,-128.817,175.200,42.043,158.283
C08873=1051.645,422.855,-128.864,175.210,42.051,158.286
C08874=1051.655,423.100,-128.911,175.220,42.061,158.289
C08875=1051.665,423.345,-128.960,175.231,42.070,158.292
C08876=1051.675,423.590,-129.007,175.240,42.079,158.295
C08877=1051.685,423.836,-129.054,175.250,42.089,158.298
C08878=1051.695,424.081,-129.102,175.261,42.098,158.302
C08879=1051.705,424.326,-129.149,175.271,42.107,158.305
C08880=1051.716,424.571,-129.197,175.281,42.117,158.308
C08881=1051.726,424.817,-129.245,175.291,42.126,158.311
C08882=1051.736,425.063,-129.293,175.302,42.135,158.314
C08883=1051.746,425.307,-129.341,175.312,42.145,158.317
C08884=1051.756,425.553,-129.388,175.323,42.154,158.321
C08885=1051.766,425.798,-129.436,175.333,42.163,158.324
C08886=1051.776,426.043,-129.485,175.344,42.173,158.327
C08887=1051.787,426.289,-129.532,175.354,42.183,158.330
C08888=1051.797,426.534,-129.581,175.365,42.192,158.334
C08889=1051.807,426.778,-129.629,175.375,42.202,158.337
C08890=1051.817,427.023,-129.677,175.386,42.211,158.340
C08891=1051.827,427.268,-129.726,175.397,42.221,158.343
C08892=1051.837,427.514,-129.774,175.407,42.231,158.347
C08893=1051.847,427.759,-129.822,175.418,42.240,158.350
C08894=1051.858,428.004,-129.870,175.429,42.250,158.353
C08895=1051.868,428.249,-129.919,175.439,42.260,158.357
C08896=1051.879,428.494,-129.968,175.450,42.270,158.360
C08897=1051.889,428.739,-130.016,175.461,42.279,158.364
C08898=1051.899,428.984,-130.065,175.472,42.289,158.367
C08899=1051.909,429.229,-130.113,175.483,42.299,158.370
C08900=1051.920,429.475,-130.162,175.494,42.309,158.374
C08901=1051.931,429.719,-130.210,175.505,42.319,158.377
C08902=1051.941,429.964,-130.259,175.516,42.329,158.381
C08903=1051.951,430.209,-130.309,175.528,42.339,158.384
C08904=1051.961,430.454,-130.357,175.539,42.349,158.388
C08905=1051.971,430.699,-130.407,175.550,42.359,158.391
C08906=1051.982,430.944,-130.456,175.560,42.369,158.395
C08907=1051.993,431.189,-130.505,175.572,42.380,158.398
C08908=1052.003,431.433,-130.554,175.583,42.390,158.402
C08909=1052.021,431.835,-130.635,175.602,42.406,158.407
C08910=1052.037,432.236,-130.715,175.621,42.423,158.413
C08911=1052.055,432.637,-130.796,175.640,42.440,158.419
C08912=1052.072,433.038,-130.877,175.659,42.457,158.425
C08913=1052.083,433.283,-130.926,175.671,42.467,158.429
C08914=1052.094,433.528,-130.977,175.682,42.478,158.433
C08915=1052.104,433.773,-131.026,175.694,42.488,158.436
C08916=1052.115,434.017,-131.075,175.705,42.499,158.440
C08917=1052.126,434.262,-131.124,175.717,42.509,158.444
C08918=1052.137,434.506,-131.175,175.729,42.519,158.447
C08919=1052.147,434.752,-131.224,175.741,42.530,158.451
C08920=1052.158,434.997,-131.274,175.753,42.541,158.455
C08921=1052.169,435.241,-131.324,175.765,42.551,158.458
C08922=1052.180,435.486,-131.374,175.777,42.562,158.462
C08923=1052.191,435.730,-131.424,175.789,42.573,158.466
C08924=1052.202,435.975,-131.473,175.802,42.583,158.470
C08925=1052.214,436.220,-131.524,175.813,42.594,158.474
C08926=1052.225,436.465,-131.574,175.826,42.605,158.478
C08927=1052.235,436.710,-131.624,175.838,42.616,158.481
C08928=1052.246,436.954,-131.674,175.850,42.627,158.485
C08929=1052.257,437.199,-131.725,175.863,42.637,158.489
C08930=1052.268,437.443,-131.775,175.876,42.648,158.493
C08931=1052.279,437.689,-131.826,175.888,42.659,158.497
C08932=1052.290,437.933,-131.876,175.901,42.670,158.501
C08933=1052.301,438.177,-131.927,175.913,42.681,158.505
C08934=1052.312,438.421,-131.978,175.925,42.692,158.509
C08935=1052.324,438.666,-132.029,175.938,42.704,158.513
C08936=1052.335,438.911,-132.079,175.951,42.715,158.517
C08937=1052.345,439.156,-132.130,175.964,42.726,158.521
C08938=1052.357,439.400,-132.181,175.977,42.737,158.525
C08939=1052.368,439.644,-132.232,175.989,42.748,158.529
C08940=1052.380,439.889,-132.283,176.002,42.760,158.533
C08941=1052.391,440.133,-132.333,176.015,42.771,158.537
C08942=1052.401,440.378,-132.385,176.028,42.783,158.541
C08943=1052.413,440.622,-132.436,176.041,42.794,158.545
C08944=1052.425,440.867,-132.488,176.054,42.806,158.550
C08945=1052.436,441.111,-132.538,176.067,42.817,158.554
C08946=1052.447,441.356,-132.590,176.080,42.828,158.558
C08947=1052.459,441.600,-132.641,176.094,42.840,158.562
C08948=1052.470,441.844,-132.692,176.107,42.851,158.566
C08949=1052.482,442.089,-132.744,176.120,42.863,158.571
C08950=1052.493,442.333,-132.795,176.134,42.874,158.575
C08951=1052.505,442.577,-132.847,176.147,42.886,158.579
C08952=1052.516,442.822,-132.899,176.161,42.898,158.583
C08953=1052.527,443.065,-132.951,176.174,42.910,158.588
C08954=1052.539,443.310,-133.002,176.188,42.922,158.592
C08955=1052.550,443.555,-133.054,176.202,42.933,158.596
C08956=1052.563,443.799,-133.106,176.216,42.945,158.601
C08957=1052.574,444.043,-133.158,176.229,42.957,158.605
C08958=1052.586,444.287,-133.210,176.243,42.969,158.609
C08959=1052.597,444.531,-133.263,176.258,42.981,158.614
C08960=1052.609,444.776,-133.314,176.271,42.993,158.618
C08961=1052.621,445.020,-133.367,176.285,43.005,158.623
C08962=1052.633,445.264,-133.419,176.300,43.017,158.627
C08963=1052.645,445.508,-133.471,176.314,43.029,158.632
C08964=1052.656,445.753,-133.523,176.327,43.041,158.636
C08965=1052.676,446.165,-133.612,176.352,43.062,158.644
C08966=1052.698,446.578,-133.700,176.376,43.082,158.652
C08967=1052.709,446.785,-133.744,176.389,43.092,158.656
C08968=1052.720,446.993,-133.787,176.401,43.102,158.659
C08969=1052.733,447.201,-133.830,176.414,43.112,158.663
C08970=1052.746,447.409,-133.872,176.426,43.122,158.667
C08971=1052.762,447.653,-133.922,176.441,43.133,158.671
C08972=1052.779,447.897,-133.970,176.456,43.144,158.676
C08973=1052.797,448.141,-134.019,176.470,43.155,158.680
C08974=1052.814,448.386,-134.067,176.485,43.166,158.684
C08975=1052.833,448.631,-134.114,176.501,43.177,158.688
C08976=1052.853,448.875,-134.160,176.515,43.187,158.693
C08977=1052.873,449.120,-134.206,176.531,43.198,158.697
C08978=1052.894,449.365,-134.252,176.546,43.208,158.701
C08979=1052.916,449.610,-134.297,176.562,43.218,158.705
C08980=1052.939,449.856,-134.342,176.577,43.227,158.709
C08981=1052.962,450.101,-134.385,176.592,43.237,158.713
C08982=1052.986,450.346,-134.429,176.608,43.246,158.717
C08983=1052.669,450.369,-134.723,176.608,43.344,158.745
C08984=1052.644,450.124,-134.680,176.591,43.334,158.741
C08985=1052.621,449.879,-134.636,176.575,43.325,158.737
C08986=1052.598,449.634,-134.592,176.560,43.315,158.733
C08987=1052.576,449.388,-134.547,176.545,43.305,158.729
C08988=1052.554,449.143,-134.502,176.530,43.295,158.725
C08989=1052.534,448.899,-134.455,176.514,43.285,158.720
C08990=1052.514,448.653,-134.409,176.499,43.274,158.716
C08991=1052.495,448.409,-134.363,176.484,43.264,158.712
C08992=1052.476,448.165,-134.314,176.468,43.253,158.708
C08993=1052.459,447.920,-134.266,176.454,43.242,158.703
C08994=1052.442,447.676,-134.217,176.439,43.231,158.699
C08995=1052.426,447.432,-134.169,176.424,43.221,158.695
C08996=1052.401,447.034,-134.086,176.400,43.202,158.688
C08997=1052.378,446.638,-134.004,176.376,43.183,158.680
C08998=1052.358,446.243,-133.920,176.353,43.163,158.673
C08999=1052.339,445.849,-133.836,176.329,43.144,158.666
C09000=1052.327,445.605,-133.783,176.315,43.132,158.661
C09001=1052.315,445.361,-133.731,176.301,43.120,158.657
C09002=1052.303,445.117,-133.679,176.287,43.108,158.652
C09003=1052.291,444.873,-133.626,176.273,43.096,158.648
C09004=1052.280,444.629,-133.575,176.258,43.084,158.643
C09005=1052.268,444.384,-133.522,176.244,43.072,158.639
C09006=1052.256,444.141,-133.470,176.231,43.060,158.634
C09007=1052.244,443.896,-133.418,176.216,43.048,158.630
C09008=1052.233,443.652,-133.366,176.202,43.036,158.625
C09009=1052.221,443.407,-133.314,176.189,43.024,158.621
C09010=1052.209,443.163,-133.261,176.175,43.013,158.617
C09011=1052.198,442.919,-133.210,176.162,43.001,158.612
C09012=1052.186,442.675,-133.159,176.148,42.989,158.608
C09013=1052.175,442.430,-133.107,176.134,42.978,158.604
C09014=1052.163,442.186,-133.055,176.120,42.966,158.599
C09015=1052.151,441.942,-133.004,176.107,42.955,158.595
C09016=1052.140,441.698,-132.952,176.094,42.943,158.591
C09017=1052.128,441.453,-132.900,176.080,42.932,158.587
C09018=1052.117,441.209,-132.849,176.067,42.921,158.583
C09019=1052.105,440.965,-132.798,176.054,42.909,158.578
C09020=1052.094,440.719,-132.747,176.041,42.898,158.574
C09021=1052.083,440.475,-132.696,176.028,42.886,158.570
C09022=1052.071,440.231,-132.644,176.015,42.875,158.566
C09023=1052.060,439.986,-132.594,176.001,42.863,158.562
C09024=1052.049,439.742,-132.542,175.988,42.853,158.558
C09025=1052.038,439.498,-132.491,175.975,42.841,158.554
C09026=1052.027,439.253,-132.441,175.963,42.830,158.550
C09027=1052.015,439.008,-132.390,175.950,42.819,158.545
C09028=1052.004,438.764,-132.339,175.937,42.808,158.541
C09029=1051.993,438.519,-132.288,175.924,42.797,158.538
C09030=1051.982,438.275,-132.237,175.912,42.786,158.534
C09031=1051.971,438.030,-132.187,175.899,42.775,158.530
C09032=1051.959,437.786,-132.136,175.887,42.764,158.526
C09033=1051.948,437.541,-132.085,175.874,42.753,158.522
C09034=1051.937,437.297,-132.035,175.861,42.742,158.518
C09035=1051.926,437.052,-131.985,175.849,42.731,158.514
C09036=1051.915,436.808,-131.934,175.836,42.720,158.510
C09037=1051.904,436.563,-131.884,175.824,42.709,158.506
C09038=1051.893,436.318,-131.834,175.811,42.699,158.502
C09039=1051.882,436.073,-131.784,175.799,42.688,158.498
C09040=1051.871,435.829,-131.733,175.787,42.677,158.494
